LIN {X 0,Y 370.334,Z 1271.38,A -85,B 0,C 180,E1 17928.905,E2 17928.905} C_VEL
LIN {X 0,Y 369.324,Z 1281.028,A -85,B 0,C 180,E1 17925.869,E2 17925.869} C_VEL
LIN {X 0,Y 368.724,Z 1288.757,A -85,B 0,C 180,E1 17922.848,E2 17922.848} C_VEL
LIN {X 0,Y 368.382,Z 1295.019,A -85,B 0,C 180,E1 17919.688,E2 17919.688} C_VEL
LIN {X 0,Y 368.28,Z 1299.31,A -85,B 0,C 180,E1 17916.705,E2 17916.705} C_VEL
LIN {X 0,Y 368.262,Z 1302.013,A -85,B 0,C 180,E1 17913.737,E2 17913.737} C_VEL
LIN {X 0,Y 368.271,Z 1303.134,A -85,B 0,C 180,E1 17910.779,E2 17910.779} C_VEL
LIN {X 0,Y 368.275,Z 1302.722,A -85,B 0,C 180,E1 17907.667,E2 17907.667} C_VEL
LIN {X 0,Y 368.252,Z 1300.81,A -85,B 0,C 180,E1 17904.704,E2 17904.704} C_VEL
LIN {X 0,Y 368.291,Z 1297.252,A -85,B 0,C 180,E1 17901.728,E2 17901.728} C_VEL
LIN {X 0,Y 368.472,Z 1292.124,A -85,B 0,C 180,E1 17898.734,E2 17898.734} C_VEL
LIN {X 0,Y 368.884,Z 1285.33,A -85,B 0,C 180,E1 17895.721,E2 17895.721} C_VEL
LIN {X 0,Y 369.628,Z 1276.713,A -85,B 0,C 180,E1 17892.69,E2 17892.69} C_VEL
LIN {X 0,Y 370.897,Z 1266.188,A -85,B 0,C 180,E1 17889.486,E2 17889.486} C_VEL
LIN {X 0,Y 372.62,Z 1254.112,A -85,B 0,C 180,E1 17886.434,E2 17886.434} C_VEL
LIN {X 0,Y 374.842,Z 1240.532,A -85,B 0,C 180,E1 17883.548,E2 17883.548} C_VEL
LIN {X 0,Y 377.687,Z 1224.468,A -85,B 0,C 180,E1 17880.677,E2 17880.677} C_VEL
LIN {X 0,Y 380.995,Z 1206.604,A -85,B 0,C 180,E1 17877.988,E2 17877.988} C_VEL
LIN {X 0,Y 384.421,Z 1188.101,A -85,B 0,C 180,E1 17875.64,E2 17875.64} C_VEL
LIN {X 0,Y 387.844,Z 1169.342,A -85,B 0,C 180,E1 17873.635,E2 17873.635} C_VEL
LIN {X 0,Y 391.563,Z 1148.3,A -85,B 0,C 180,E1 17871.741,E2 17871.741} C_VEL
LIN {X 0,Y 394.879,Z 1128.554,A -85,B 0,C 180,E1 17870.258,E2 17870.258} C_VEL
LIN {X 0,Y 398.329,Z 1105.945,A -85,B 0,C 180,E1 17868.88,E2 17868.88} C_VEL
LIN {X 0,Y 401.441,Z 1082.847,A -85,B 0,C 180,E1 17867.777,E2 17867.777} C_VEL
LIN {X 0,Y 404.065,Z 1059.287,A -85,B 0,C 180,E1 17866.948,E2 17866.948} C_VEL
LIN {X 0,Y 405.779,Z 1035.371,A -85,B 0,C 180,E1 17866.328,E2 17866.328} C_VEL
LIN {X 0,Y 407.409,Z 1016.443,A -85,B 0,C 180,E1 17865.98,E2 17865.98} C_VEL
LIN {X 0,Y 408.442,Z 1008.559,A -85,B 0,C 180,E1 17865.858,E2 17865.858} C_VEL
LIN {X 0,Y 420.821,Z 978.098,A -85,B 0,C 180,E1 17864.422,E2 17864.422} C_VEL
LIN {X 0,Y 430.29,Z 959.013,A -85,B 0,C 180,E1 17863.726,E2 17863.726} C_VEL
LIN {X 0,Y 442.106,Z 935.256,A -85,B 0,C 180,E1 17862.901,E2 17862.901} C_VEL
LIN {X 0,Y 444.175,Z 931.152,A -85,B 0,C 180,E1 17862.767,E2 17862.767} C_VEL
LIN {X 0,Y 436.092,Z 918.557,A -85,B 0,C 180,E1 17860.801,E2 17860.801} C_VEL
LIN {X 0,Y 429.406,Z 903.824,A -85,B 0,C 180,E1 17858.696,E2 17858.696} C_VEL
LIN {X 0,Y 424.66,Z 887.722,A -85,B 0,C 180,E1 17856.595,E2 17856.595} C_VEL
LIN {X 0,Y 421.837,Z 870.153,A -85,B 0,C 180,E1 17854.505,E2 17854.505} C_VEL
LIN {X 0,Y 420.994,Z 850.406,A -85,B 0,C 180,E1 17852.382,E2 17852.382} C_VEL
LIN {X 0,Y 422.168,Z 830.506,A -85,B 0,C 180,E1 17850.449,E2 17850.449} C_VEL
LIN {X 0,Y 426.561,Z 800.035,A -85,B 0,C 180,E1 17847.804,E2 17847.804} C_VEL
LIN {X 0,Y 427.695,Z 792.967,A -85,B 0,C 180,E1 17847.196,E2 17847.196} C_VEL
LIN {X 0,Y 418.747,Z 775.54,A -85,B 0,C 180,E1 17843.649,E2 17843.649} C_VEL
LIN {X 0,Y 409.719,Z 758.616,A -85,B 0,C 180,E1 17839.828,E2 17839.828} C_VEL
LIN {X 0,Y 401.65,Z 744.073,A -85,B 0,C 180,E1 17836.189,E2 17836.189} C_VEL
LIN {X 0,Y 395.059,Z 732.588,A -85,B 0,C 180,E1 17833.017,E2 17833.017} C_VEL
LIN {X 0,Y 390.083,Z 723.936,A -85,B 0,C 180,E1 17830.485,E2 17830.485} C_VEL
LIN {X 0,Y 387.124,Z 718.9,A -85,B 0,C 180,E1 17828.915,E2 17828.915} C_VEL
LIN {X 0,Y 384.512,Z 714.317,A -85,B 0,C 180,E1 17827.47,E2 17827.47} C_VEL
LIN {X 0,Y 381.689,Z 709.437,A -85,B 0,C 180,E1 17825.863,E2 17825.863} C_VEL
LIN {X 0,Y 379.41,Z 705.573,A -85,B 0,C 180,E1 17824.534,E2 17824.534} C_VEL
LIN {X 0,Y 378.063,Z 703.576,A -85,B 0,C 180,E1 17823.791,E2 17823.791} C_VEL
LIN {X 0,Y 375.728,Z 699.193,A -85,B 0,C 180,E1 17822.287,E2 17822.287} C_VEL
LIN {X 0,Y 373.418,Z 695.781,A -85,B 0,C 180,E1 17820.92,E2 17820.92} C_VEL
LIN {X 0,Y 372.606,Z 693.864,A -85,B 0,C 180,E1 17820.307,E2 17820.307} C_VEL
LIN {X 0,Y 370.262,Z 690.693,A -85,B 0,C 180,E1 17818.917,E2 17818.917} C_VEL
LIN {X 0,Y 369.747,Z 688.673,A -85,B 0,C 180,E1 17818.295,E2 17818.295} C_VEL
LIN {X 0,Y 369.749,Z 688.674,A -85,B 0,C 180,E1 17814.102,E2 17814.102} C_VEL
LIN {X 0,Y 369.75,Z 688.677,A -85,B 0,C 180,E1 17809.876,E2 17809.876} C_VEL
LIN {X 0,Y 369.748,Z 688.678,A -85,B 0,C 180,E1 17805.754,E2 17805.754} C_VEL
LIN {X 0,Y 369.737,Z 688.666,A -85,B 0,C 180,E1 17801.654,E2 17801.654} C_VEL
LIN {X 0,Y 369.739,Z 688.667,A -85,B 0,C 180,E1 17797.586,E2 17797.586} C_VEL
LIN {X 0,Y 369.743,Z 688.647,A -85,B 0,C 180,E1 17793.5,E2 17793.5} C_VEL
LIN {X 0,Y 369.739,Z 688.661,A -85,B 0,C 180,E1 17789.674,E2 17789.674} C_VEL
LIN {X 0,Y 370.97,Z 692.001,A -85,B 0,C 180,E1 17788.99,E2 17788.99} C_VEL
LIN {X 0,Y 373.172,Z 694.719,A -85,B 0,C 180,E1 17788.14,E2 17788.14} C_VEL
LIN {X 0,Y 375.236,Z 698.459,A -85,B 0,C 180,E1 17787.254,E2 17787.254} C_VEL
LIN {X 0,Y 376.535,Z 700.304,A -85,B 0,C 180,E1 17786.766,E2 17786.766} C_VEL
LIN {X 0,Y 382.225,Z 710.075,A -85,B 0,C 180,E1 17784.498,E2 17784.498} C_VEL
LIN {X 0,Y 389.28,Z 723.15,A -85,B 0,C 180,E1 17781.756,E2 17781.756} C_VEL
LIN {X 0,Y 396.449,Z 737.875,A -85,B 0,C 180,E1 17779.025,E2 17779.025} C_VEL
LIN {X 0,Y 403.876,Z 755.101,A -85,B 0,C 180,E1 17776.215,E2 17776.215} C_VEL
LIN {X 0,Y 407.155,Z 763.877,A -85,B 0,C 180,E1 17774.938,E2 17774.938} C_VEL
LIN {X 0,Y 406.421,Z 778.004,A -85,B 0,C 180,E1 17773.911,E2 17773.911} C_VEL
LIN {X 0,Y 409.717,Z 805.43,A -85,B 0,C 180,E1 17772.811,E2 17772.811} C_VEL
LIN {X 0,Y 401.369,Z 1038.951,A -85,B 0,C 180,E1 17768.404,E2 17768.404} C_VEL
LIN {X 0,Y 400.003,Z 1059.693,A -85,B 0,C 180,E1 17767.771,E2 17767.771} C_VEL
LIN {X 0,Y 398.071,Z 1079.901,A -85,B 0,C 180,E1 17766.891,E2 17766.891} C_VEL
LIN {X 0,Y 395.711,Z 1098.998,A -85,B 0,C 180,E1 17765.798,E2 17765.798} C_VEL
LIN {X 0,Y 392.961,Z 1117.404,A -85,B 0,C 180,E1 17764.473,E2 17764.473} C_VEL
LIN {X 0,Y 389.794,Z 1135.566,A -85,B 0,C 180,E1 17762.854,E2 17762.854} C_VEL
LIN {X 0,Y 386.595,Z 1152.047,A -85,B 0,C 180,E1 17761.061,E2 17761.061} C_VEL
LIN {X 0,Y 383.311,Z 1167.686,A -85,B 0,C 180,E1 17759.023,E2 17759.023} C_VEL
LIN {X 0,Y 380.099,Z 1182.367,A -85,B 0,C 180,E1 17756.731,E2 17756.731} C_VEL
LIN {X 0,Y 377.097,Z 1195.87,A -85,B 0,C 180,E1 17754.202,E2 17754.202} C_VEL
LIN {X 0,Y 376.683,Z 1197.706,A -85,B 0,C 180,E1 17753.819,E2 17753.819} C_VEL
LIN {X 0,Y 374.766,Z 1202.283,A -85,B 0,C 180,E1 17752.903,E2 17752.903} C_VEL
LIN {X 0,Y 366.788,Z 1213.338,A -85,B 0,C 180,E1 17750.607,E2 17750.607} C_VEL
LIN {X 0,Y 365.037,Z 1217.109,A -85,B 0,C 180,E1 17749.588,E2 17749.588} C_VEL
LIN {X 0,Y 363.2,Z 1226.026,A -85,B 0,C 180,E1 17746.636,E2 17746.636} C_VEL
LIN {X 0,Y 361.799,Z 1233.817,A -85,B 0,C 180,E1 17743.398,E2 17743.398} C_VEL
LIN {X 0,Y 360.949,Z 1239.677,A -85,B 0,C 180,E1 17740.211,E2 17740.211} C_VEL
LIN {X 0,Y 360.49,Z 1243.91,A -85,B 0,C 180,E1 17737.009,E2 17737.009} C_VEL
LIN {X 0,Y 360.28,Z 1246.508,A -85,B 0,C 180,E1 17733.818,E2 17733.818} C_VEL
LIN {X 0,Y 360.214,Z 1247.557,A -85,B 0,C 180,E1 17730.635,E2 17730.635} C_VEL
LIN {X 0,Y 360.238,Z 1247.128,A -85,B 0,C 180,E1 17727.454,E2 17727.454} C_VEL
LIN {X 0,Y 360.371,Z 1245.21,A -85,B 0,C 180,E1 17724.267,E2 17724.267} C_VEL
LIN {X 0,Y 360.714,Z 1241.72,A -85,B 0,C 180,E1 17721.069,E2 17721.069} C_VEL
LIN {X 0,Y 361.39,Z 1236.528,A -85,B 0,C 180,E1 17717.861,E2 17717.861} C_VEL
LIN {X 0,Y 362.462,Z 1229.973,A -85,B 0,C 180,E1 17714.807,E2 17714.807} C_VEL
LIN {X 0,Y 364.176,Z 1221.194,A -85,B 0,C 180,E1 17711.594,E2 17711.594} C_VEL
LIN {X 0,Y 366.437,Z 1210.813,A -85,B 0,C 180,E1 17708.553,E2 17708.553} C_VEL
LIN {X 0,Y 369.026,Z 1199.594,A -85,B 0,C 180,E1 17705.849,E2 17705.849} C_VEL
LIN {X 0,Y 371.993,Z 1187.057,A -85,B 0,C 180,E1 17703.328,E2 17703.328} C_VEL
LIN {X 0,Y 375.48,Z 1172.083,A -85,B 0,C 180,E1 17700.836,E2 17700.836} C_VEL
LIN {X 0,Y 378.941,Z 1156.452,A -85,B 0,C 180,E1 17698.681,E2 17698.681} C_VEL
LIN {X 0,Y 382.302,Z 1140.187,A -85,B 0,C 180,E1 17696.816,E2 17696.816} C_VEL
LIN {X 0,Y 385.626,Z 1122.381,A -85,B 0,C 180,E1 17695.129,E2 17695.129} C_VEL
LIN {X 0,Y 388.618,Z 1104.067,A -85,B 0,C 180,E1 17693.718,E2 17693.718} C_VEL
LIN {X 0,Y 391.179,Z 1085.559,A -85,B 0,C 180,E1 17692.575,E2 17692.575} C_VEL
LIN {X 0,Y 393.361,Z 1065.157,A -85,B 0,C 180,E1 17691.604,E2 17691.604} C_VEL
LIN {X 0,Y 394.969,Z 1043.732,A -85,B 0,C 180,E1 17690.883,E2 17690.883} C_VEL
LIN {X 0,Y 396.204,Z 1013.325,A -85,B 0,C 180,E1 17690.248,E2 17690.248} C_VEL
LIN {X 0,Y 403.433,Z 816.76,A -85,B 0,C 180,E1 17686.515,E2 17686.515} C_VEL
LIN {X 0,Y 395.988,Z 779.414,A -85,B 0,C 180,E1 17684.495,E2 17684.495} C_VEL
LIN {X 0,Y 396.639,Z 768.209,A -85,B 0,C 180,E1 17683.237,E2 17683.237} C_VEL
LIN {X 0,Y 394.121,Z 760.718,A -85,B 0,C 180,E1 17681.853,E2 17681.853} C_VEL
LIN {X 0,Y 393.361,Z 760.544,A -85,B 0,C 180,E1 17681.642,E2 17681.642} C_VEL
LIN {X 0,Y 394.85,Z 764.717,A -85,B 0,C 180,E1 17680.898,E2 17680.898} C_VEL
LIN {X 0,Y 389.829,Z 803.215,A -85,B 0,C 180,E1 17676.8,E2 17676.8} C_VEL
LIN {X 0,Y 385.068,Z 843.255,A -85,B 0,C 180,E1 17672.602,E2 17672.602} C_VEL
LIN {X 0,Y 382.539,Z 867.952,A -85,B 0,C 180,E1 17670.081,E2 17670.081} C_VEL
LIN {X 0,Y 383.563,Z 877.843,A -85,B 0,C 180,E1 17669.684,E2 17669.684} C_VEL
LIN {X 0,Y 375.672,Z 1037.088,A -85,B 0,C 180,E1 17665.526,E2 17665.526} C_VEL
LIN {X 0,Y 374.898,Z 1054.189,A -85,B 0,C 180,E1 17664.838,E2 17664.838} C_VEL
LIN {X 0,Y 373.669,Z 1071.817,A -85,B 0,C 180,E1 17663.832,E2 17663.832} C_VEL
LIN {X 0,Y 372.206,Z 1088.344,A -85,B 0,C 180,E1 17662.591,E2 17662.591} C_VEL
LIN {X 0,Y 370.57,Z 1103.821,A -85,B 0,C 180,E1 17661.113,E2 17661.113} C_VEL
LIN {X 0,Y 368.793,Z 1118.857,A -85,B 0,C 180,E1 17659.315,E2 17659.315} C_VEL
LIN {X 0,Y 367.142,Z 1131.984,A -85,B 0,C 180,E1 17657.39,E2 17657.39} C_VEL
LIN {X 0,Y 365.594,Z 1143.989,A -85,B 0,C 180,E1 17655.222,E2 17655.222} C_VEL
LIN {X 0,Y 364.239,Z 1154.622,A -85,B 0,C 180,E1 17652.847,E2 17652.847} C_VEL
LIN {X 0,Y 363.188,Z 1163.735,A -85,B 0,C 180,E1 17650.309,E2 17650.309} C_VEL
LIN {X 0,Y 362.494,Z 1170.776,A -85,B 0,C 180,E1 17647.768,E2 17647.768} C_VEL
LIN {X 0,Y 362.034,Z 1176.672,A -85,B 0,C 180,E1 17644.912,E2 17644.912} C_VEL
LIN {X 0,Y 361.881,Z 1180.442,A -85,B 0,C 180,E1 17642.217,E2 17642.217} C_VEL
LIN {X 0,Y 361.917,Z 1182.564,A -85,B 0,C 180,E1 17639.367,E2 17639.367} C_VEL
LIN {X 0,Y 362.162,Z 1182.94,A -85,B 0,C 180,E1 17636.518,E2 17636.518} C_VEL
LIN {X 0,Y 362.626,Z 1181.617,A -85,B 0,C 180,E1 17633.827,E2 17633.827} C_VEL
LIN {X 0,Y 363.414,Z 1178.412,A -85,B 0,C 180,E1 17630.978,E2 17630.978} C_VEL
LIN {X 0,Y 364.517,Z 1173.647,A -85,B 0,C 180,E1 17628.289,E2 17628.289} C_VEL
LIN {X 0,Y 366.041,Z 1166.884,A -85,B 0,C 180,E1 17625.607,E2 17625.607} C_VEL
LIN {X 0,Y 367.931,Z 1158.574,A -85,B 0,C 180,E1 17623.096,E2 17623.096} C_VEL
LIN {X 0,Y 370.08,Z 1148.58,A -85,B 0,C 180,E1 17620.755,E2 17620.755} C_VEL
LIN {X 0,Y 372.266,Z 1137.95,A -85,B 0,C 180,E1 17618.741,E2 17618.741} C_VEL
LIN {X 0,Y 374.503,Z 1125.805,A -85,B 0,C 180,E1 17616.892,E2 17616.892} C_VEL
LIN {X 0,Y 376.769,Z 1112.27,A -85,B 0,C 180,E1 17615.21,E2 17615.21} C_VEL
LIN {X 0,Y 379.043,Z 1095.883,A -85,B 0,C 180,E1 17613.61,E2 17613.61} C_VEL
LIN {X 0,Y 380.683,Z 1080.836,A -85,B 0,C 180,E1 17612.467,E2 17612.467} C_VEL
LIN {X 0,Y 382.09,Z 1064.158,A -85,B 0,C 180,E1 17611.495,E2 17611.495} C_VEL
LIN {X 0,Y 385.237,Z 1037.1,A -85,B 0,C 180,E1 17610.154,E2 17610.154} C_VEL
LIN {X 0,Y 394.185,Z 989.779,A -85,B 0,C 180,E1 17607.986,E2 17607.986} C_VEL
LIN {X 0,Y 405.123,Z 935.467,A -85,B 0,C 180,E1 17605.776,E2 17605.776} C_VEL
LIN {X 0,Y 406.823,Z 928.336,A -85,B 0,C 180,E1 17605.494,E2 17605.494} C_VEL
LIN {X 0,Y 417.353,Z 912.085,A -85,B 0,C 180,E1 17604.482,E2 17604.482} C_VEL
LIN {X 0,Y 423.503,Z 903.048,A -85,B 0,C 180,E1 17603.827,E2 17603.827} C_VEL
LIN {X 0,Y 426.01,Z 899.819,A -85,B 0,C 180,E1 17603.301,E2 17603.301} C_VEL
LIN {X 0,Y 424.14,Z 907.115,A -85,B 0,C 180,E1 17601.504,E2 17601.504} C_VEL
LIN {X 0,Y 424.485,Z 914.511,A -85,B 0,C 180,E1 17599.745,E2 17599.745} C_VEL
LIN {X 0,Y 427.026,Z 922.456,A -85,B 0,C 180,E1 17597.96,E2 17597.96} C_VEL
LIN {X 0,Y 430.407,Z 928.617,A -85,B 0,C 180,E1 17596.646,E2 17596.646} C_VEL
LIN {X 0,Y 420.892,Z 947.99,A -85,B 0,C 180,E1 17595.97,E2 17595.97} C_VEL
LIN {X 0,Y 409.338,Z 971.916,A -85,B 0,C 180,E1 17595.102,E2 17595.102} C_VEL
LIN {X 0,Y 407.173,Z 977.442,A -85,B 0,C 180,E1 17594.891,E2 17594.891} C_VEL
LIN {X 0,Y 403.741,Z 996.518,A -85,B 0,C 180,E1 17594.623,E2 17594.623} C_VEL
LIN {X 0,Y 399.024,Z 1022.37,A -85,B 0,C 180,E1 17594.225,E2 17594.225} C_VEL
LIN {X 0,Y 396.381,Z 1040.88,A -85,B 0,C 180,E1 17593.63,E2 17593.63} C_VEL
LIN {X 0,Y 392.042,Z 1070.576,A -85,B 0,C 180,E1 17592.381,E2 17592.381} C_VEL
LIN {X 0,Y 387.903,Z 1096.54,A -85,B 0,C 180,E1 17590.996,E2 17590.996} C_VEL
LIN {X 0,Y 383.805,Z 1122.59,A -85,B 0,C 180,E1 17589.276,E2 17589.276} C_VEL
LIN {X 0,Y 379.789,Z 1149.026,A -85,B 0,C 180,E1 17587.208,E2 17587.208} C_VEL
LIN {X 0,Y 377.55,Z 1169.051,A -85,B 0,C 180,E1 17585.608,E2 17585.608} C_VEL
LIN {X 0,Y 375.105,Z 1187.196,A -85,B 0,C 180,E1 17583.856,E2 17583.856} C_VEL
LIN {X 0,Y 372.581,Z 1204.537,A -85,B 0,C 180,E1 17581.849,E2 17581.849} C_VEL
LIN {X 0,Y 370.039,Z 1220.672,A -85,B 0,C 180,E1 17579.636,E2 17579.636} C_VEL
LIN {X 0,Y 367.548,Z 1236.156,A -85,B 0,C 180,E1 17577.108,E2 17577.108} C_VEL
LIN {X 0,Y 365.512,Z 1249.285,A -85,B 0,C 180,E1 17574.57,E2 17574.57} C_VEL
LIN {X 0,Y 363.66,Z 1261.967,A -85,B 0,C 180,E1 17571.674,E2 17571.674} C_VEL
LIN {X 0,Y 362.251,Z 1272.901,A -85,B 0,C 180,E1 17568.674,E2 17568.674} C_VEL
LIN {X 0,Y 361.25,Z 1282.119,A -85,B 0,C 180,E1 17565.596,E2 17565.596} C_VEL
LIN {X 0,Y 360.683,Z 1289.596,A -85,B 0,C 180,E1 17562.488,E2 17562.488} C_VEL
LIN {X 0,Y 360.371,Z 1295.202,A -85,B 0,C 180,E1 17559.422,E2 17559.422} C_VEL
LIN {X 0,Y 360.293,Z 1299.202,A -85,B 0,C 180,E1 17556.374,E2 17556.374} C_VEL
LIN {X 0,Y 360.282,Z 1301.681,A -85,B 0,C 180,E1 17553.342,E2 17553.342} C_VEL
LIN {X 0,Y 360.297,Z 1302.595,A -85,B 0,C 180,E1 17550.319,E2 17550.319} C_VEL
LIN {X 0,Y 360.286,Z 1301.969,A -85,B 0,C 180,E1 17547.297,E2 17547.297} C_VEL
LIN {X 0,Y 360.267,Z 1299.87,A -85,B 0,C 180,E1 17544.267,E2 17544.267} C_VEL
LIN {X 0,Y 360.317,Z 1296.202,A -85,B 0,C 180,E1 17541.222,E2 17541.222} C_VEL
LIN {X 0,Y 360.532,Z 1290.87,A -85,B 0,C 180,E1 17538.158,E2 17538.158} C_VEL
LIN {X 0,Y 361.041,Z 1283.439,A -85,B 0,C 180,E1 17534.912,E2 17534.912} C_VEL
LIN {X 0,Y 361.915,Z 1274.491,A -85,B 0,C 180,E1 17531.81,E2 17531.81} C_VEL
LIN {X 0,Y 363.181,Z 1264.14,A -85,B 0,C 180,E1 17528.861,E2 17528.861} C_VEL
LIN {X 0,Y 365.064,Z 1251.734,A -85,B 0,C 180,E1 17525.744,E2 17525.744} C_VEL
LIN {X 0,Y 367.443,Z 1237.859,A -85,B 0,C 180,E1 17522.798,E2 17522.798} C_VEL
LIN {X 0,Y 370.298,Z 1222.447,A -85,B 0,C 180,E1 17520.032,E2 17520.032} C_VEL
LIN {X 0,Y 373.687,Z 1204.93,A -85,B 0,C 180,E1 17517.376,E2 17517.376} C_VEL
LIN {X 0,Y 377.164,Z 1186.99,A -85,B 0,C 180,E1 17515.068,E2 17515.068} C_VEL
LIN {X 0,Y 380.722,Z 1168.184,A -85,B 0,C 180,E1 17513.031,E2 17513.031} C_VEL
LIN {X 0,Y 384.556,Z 1147.378,A -85,B 0,C 180,E1 17511.134,E2 17511.134} C_VEL
LIN {X 0,Y 388.053,Z 1127.311,A -85,B 0,C 180,E1 17509.609,E2 17509.609} C_VEL
LIN {X 0,Y 391.691,Z 1104.318,A -85,B 0,C 180,E1 17508.191,E2 17508.191} C_VEL
LIN {X 0,Y 394.935,Z 1081.232,A -85,B 0,C 180,E1 17507.084,E2 17507.084} C_VEL
LIN {X 0,Y 397.625,Z 1057.81,A -85,B 0,C 180,E1 17506.252,E2 17506.252} C_VEL
LIN {X 0,Y 399.394,Z 1033.97,A -85,B 0,C 180,E1 17505.622,E2 17505.622} C_VEL
LIN {X 0,Y 401.317,Z 1013.867,A -85,B 0,C 180,E1 17505.26,E2 17505.26} C_VEL
LIN {X 0,Y 402.28,Z 1007.289,A -85,B 0,C 180,E1 17505.151,E2 17505.151} C_VEL
LIN {X 0,Y 414.92,Z 976.742,A -85,B 0,C 180,E1 17503.704,E2 17503.704} C_VEL
LIN {X 0,Y 424.534,Z 957.541,A -85,B 0,C 180,E1 17503.007,E2 17503.007} C_VEL
LIN {X 0,Y 436.362,Z 933.76,A -85,B 0,C 180,E1 17502.172,E2 17502.172} C_VEL
LIN {X 0,Y 428.84,Z 921.197,A -85,B 0,C 180,E1 17500.228,E2 17500.228} C_VEL
LIN {X 0,Y 422.391,Z 906.03,A -85,B 0,C 180,E1 17498.071,E2 17498.071} C_VEL
LIN {X 0,Y 417.987,Z 889.853,A -85,B 0,C 180,E1 17495.962,E2 17495.962} C_VEL
LIN {X 0,Y 415.477,Z 872.42,A -85,B 0,C 180,E1 17493.877,E2 17493.877} C_VEL
LIN {X 0,Y 414.883,Z 852.273,A -85,B 0,C 180,E1 17491.693,E2 17491.693} C_VEL
LIN {X 0,Y 416.372,Z 830.958,A -85,B 0,C 180,E1 17489.625,E2 17489.625} C_VEL
LIN {X 0,Y 421.545,Z 797.164,A -85,B 0,C 180,E1 17486.672,E2 17486.672} C_VEL
LIN {X 0,Y 413.058,Z 780.548,A -85,B 0,C 180,E1 17483.238,E2 17483.238} C_VEL
LIN {X 0,Y 404.386,Z 764.152,A -85,B 0,C 180,E1 17479.499,E2 17479.499} C_VEL
LIN {X 0,Y 396.616,Z 750.067,A -85,B 0,C 180,E1 17475.949,E2 17475.949} C_VEL
LIN {X 0,Y 388.955,Z 736.37,A -85,B 0,C 180,E1 17472.168,E2 17472.168} C_VEL
LIN {X 0,Y 382.323,Z 725.17,A -85,B 0,C 180,E1 17468.724,E2 17468.724} C_VEL
LIN {X 0,Y 379.43,Z 720.187,A -85,B 0,C 180,E1 17467.114,E2 17467.114} C_VEL
LIN {X 0,Y 376.591,Z 715.31,A -85,B 0,C 180,E1 17465.484,E2 17465.484} C_VEL
LIN {X 0,Y 373.763,Z 710.423,A -85,B 0,C 180,E1 17463.802,E2 17463.802} C_VEL
LIN {X 0,Y 371.379,Z 706.208,A -85,B 0,C 180,E1 17462.314,E2 17462.314} C_VEL
LIN {X 0,Y 368.581,Z 701.852,A -85,B 0,C 180,E1 17460.621,E2 17460.621} C_VEL
LIN {X 0,Y 367.696,Z 700.08,A -85,B 0,C 180,E1 17460,E2 17460} C_VEL
LIN {X 0,Y 365.419,Z 696.703,A -85,B 0,C 180,E1 17458.589,E2 17458.589} C_VEL
LIN {X 0,Y 364.65,Z 694.844,A -85,B 0,C 180,E1 17457.957,E2 17457.957} C_VEL
LIN {X 0,Y 362.53,Z 692.14,A -85,B 0,C 180,E1 17456.679,E2 17456.679} C_VEL
LIN {X 0,Y 361.799,Z 689.663,A -85,B 0,C 180,E1 17455.879,E2 17455.879} C_VEL
LIN {X 0,Y 361.805,Z 689.663,A -85,B 0,C 180,E1 17451.737,E2 17451.737} C_VEL
LIN {X 0,Y 361.81,Z 689.666,A -85,B 0,C 180,E1 17447.552,E2 17447.552} C_VEL
LIN {X 0,Y 361.808,Z 689.665,A -85,B 0,C 180,E1 17443.462,E2 17443.462} C_VEL
LIN {X 0,Y 361.816,Z 689.664,A -85,B 0,C 180,E1 17439.115,E2 17439.115} C_VEL
LIN {X 0,Y 361.806,Z 689.668,A -85,B 0,C 180,E1 17434.987,E2 17434.987} C_VEL
LIN {X 0,Y 361.81,Z 689.637,A -85,B 0,C 180,E1 17431.619,E2 17431.619} C_VEL
LIN {X 0,Y 362.81,Z 692.621,A -85,B 0,C 180,E1 17430.985,E2 17430.985} C_VEL
LIN {X 0,Y 365.352,Z 695.631,A -85,B 0,C 180,E1 17429.946,E2 17429.946} C_VEL
LIN {X 0,Y 367.29,Z 699.312,A -85,B 0,C 180,E1 17429.035,E2 17429.035} C_VEL
LIN {X 0,Y 368.771,Z 701.272,A -85,B 0,C 180,E1 17428.447,E2 17428.447} C_VEL
LIN {X 0,Y 371.173,Z 705.302,A -85,B 0,C 180,E1 17427.401,E2 17427.401} C_VEL
LIN {X 0,Y 377.304,Z 715.803,A -85,B 0,C 180,E1 17424.896,E2 17424.896} C_VEL
LIN {X 0,Y 384.252,Z 728.889,A -85,B 0,C 180,E1 17422.113,E2 17422.113} C_VEL
LIN {X 0,Y 391.319,Z 743.645,A -85,B 0,C 180,E1 17419.341,E2 17419.341} C_VEL
LIN {X 0,Y 398.456,Z 760.469,A -85,B 0,C 180,E1 17416.563,E2 17416.563} C_VEL
LIN {X 0,Y 401.144,Z 767.307,A -85,B 0,C 180,E1 17415.541,E2 17415.541} C_VEL
LIN {X 0,Y 400.564,Z 778.616,A -85,B 0,C 180,E1 17414.72,E2 17414.72} C_VEL
LIN {X 0,Y 403.859,Z 806.865,A -85,B 0,C 180,E1 17413.563,E2 17413.563} C_VEL
LIN {X 0,Y 395.135,Z 1039.668,A -85,B 0,C 180,E1 17409.119,E2 17409.119} C_VEL
LIN {X 0,Y 393.72,Z 1060.288,A -85,B 0,C 180,E1 17408.481,E2 17408.481} C_VEL
LIN {X 0,Y 391.63,Z 1081.191,A -85,B 0,C 180,E1 17407.556,E2 17407.556} C_VEL
LIN {X 0,Y 389.087,Z 1100.679,A -85,B 0,C 180,E1 17406.413,E2 17406.413} C_VEL
LIN {X 0,Y 386.237,Z 1118.798,A -85,B 0,C 180,E1 17405.077,E2 17405.077} C_VEL
LIN {X 0,Y 382.934,Z 1136.929,A -85,B 0,C 180,E1 17403.43,E2 17403.43} C_VEL
LIN {X 0,Y 379.467,Z 1153.947,A -85,B 0,C 180,E1 17401.535,E2 17401.535} C_VEL
LIN {X 0,Y 375.979,Z 1169.684,A -85,B 0,C 180,E1 17399.419,E2 17399.419} C_VEL
LIN {X 0,Y 372.697,Z 1183.874,A -85,B 0,C 180,E1 17397.133,E2 17397.133} C_VEL
LIN {X 0,Y 369.628,Z 1196.944,A -85,B 0,C 180,E1 17394.618,E2 17394.618} C_VEL
LIN {X 0,Y 366.923,Z 1208.631,A -85,B 0,C 180,E1 17391.92,E2 17391.92} C_VEL
LIN {X 0,Y 365.037,Z 1217.109,A -85,B 0,C 180,E1 17389.588,E2 17389.588} C_VEL
LIN {X 0,Y 363.336,Z 1220.757,A -85,B 0,C 180,E1 17388.543,E2 17388.543} C_VEL
LIN {X 0,Y 355.548,Z 1229.785,A -85,B 0,C 180,E1 17385.732,E2 17385.732} C_VEL
LIN {X 0,Y 354.378,Z 1232.205,A -85,B 0,C 180,E1 17384.751,E2 17384.751} C_VEL
LIN {X 0,Y 353.31,Z 1238.42,A -85,B 0,C 180,E1 17381.59,E2 17381.59} C_VEL
LIN {X 0,Y 352.675,Z 1243.194,A -85,B 0,C 180,E1 17378.313,E2 17378.313} C_VEL
LIN {X 0,Y 352.365,Z 1246.365,A -85,B 0,C 180,E1 17375.046,E2 17375.046} C_VEL
LIN {X 0,Y 352.249,Z 1248.015,A -85,B 0,C 180,E1 17371.789,E2 17371.789} C_VEL
LIN {X 0,Y 352.24,Z 1248.094,A -85,B 0,C 180,E1 17368.698,E2 17368.698} C_VEL
LIN {X 0,Y 352.333,Z 1246.751,A -85,B 0,C 180,E1 17365.442,E2 17365.442} C_VEL
LIN {X 0,Y 352.598,Z 1243.897,A -85,B 0,C 180,E1 17362.176,E2 17362.176} C_VEL
LIN {X 0,Y 353.177,Z 1239.448,A -85,B 0,C 180,E1 17358.9,E2 17358.9} C_VEL
LIN {X 0,Y 354.268,Z 1232.889,A -85,B 0,C 180,E1 17355.452,E2 17355.452} C_VEL
LIN {X 0,Y 355.898,Z 1224.699,A -85,B 0,C 180,E1 17352.168,E2 17352.168} C_VEL
LIN {X 0,Y 357.954,Z 1215.506,A -85,B 0,C 180,E1 17349.222,E2 17349.222} C_VEL
LIN {X 0,Y 360.624,Z 1204.375,A -85,B 0,C 180,E1 17346.295,E2 17346.295} C_VEL
LIN {X 0,Y 363.755,Z 1191.754,A -85,B 0,C 180,E1 17343.557,E2 17343.557} C_VEL
LIN {X 0,Y 367.123,Z 1178.085,A -85,B 0,C 180,E1 17341.09,E2 17341.09} C_VEL
LIN {X 0,Y 370.751,Z 1162.946,A -85,B 0,C 180,E1 17338.815,E2 17338.815} C_VEL
LIN {X 0,Y 374.358,Z 1146.839,A -85,B 0,C 180,E1 17336.802,E2 17336.802} C_VEL
LIN {X 0,Y 377.876,Z 1129.474,A -85,B 0,C 180,E1 17335.018,E2 17335.018} C_VEL
LIN {X 0,Y 381.026,Z 1111.837,A -85,B 0,C 180,E1 17333.532,E2 17333.532} C_VEL
LIN {X 0,Y 383.894,Z 1093.135,A -85,B 0,C 180,E1 17332.261,E2 17332.261} C_VEL
LIN {X 0,Y 386.353,Z 1073.22,A -85,B 0,C 180,E1 17331.204,E2 17331.204} C_VEL
LIN {X 0,Y 388.177,Z 1053.47,A -85,B 0,C 180,E1 17330.423,E2 17330.423} C_VEL
LIN {X 0,Y 389.395,Z 1032.495,A -85,B 0,C 180,E1 17329.859,E2 17329.859} C_VEL
LIN {X 0,Y 397.671,Z 818.699,A -85,B 0,C 180,E1 17325.76,E2 17325.76} C_VEL
LIN {X 0,Y 390.082,Z 780.319,A -85,B 0,C 180,E1 17323.642,E2 17323.642} C_VEL
LIN {X 0,Y 390.524,Z 772.221,A -85,B 0,C 180,E1 17322.725,E2 17322.725} C_VEL
LIN {X 0,Y 388.925,Z 767.404,A -85,B 0,C 180,E1 17321.846,E2 17321.846} C_VEL
LIN {X 0,Y 387.838,Z 767.062,A -85,B 0,C 180,E1 17321.594,E2 17321.594} C_VEL
LIN {X 0,Y 388.24,Z 768.475,A -85,B 0,C 180,E1 17321.354,E2 17321.354} C_VEL
LIN {X 0,Y 382.997,Z 806.806,A -85,B 0,C 180,E1 17317.227,E2 17317.227} C_VEL
LIN {X 0,Y 378.087,Z 846.622,A -85,B 0,C 180,E1 17313.009,E2 17313.009} C_VEL
LIN {X 0,Y 375.688,Z 868.914,A -85,B 0,C 180,E1 17310.705,E2 17310.705} C_VEL
LIN {X 0,Y 376.687,Z 879.138,A -85,B 0,C 180,E1 17310.287,E2 17310.287} C_VEL
LIN {X 0,Y 368.367,Z 1037.296,A -85,B 0,C 180,E1 17306.029,E2 17306.029} C_VEL
LIN {X 0,Y 367.511,Z 1055.436,A -85,B 0,C 180,E1 17305.286,E2 17305.286} C_VEL
LIN {X 0,Y 366.228,Z 1073.122,A -85,B 0,C 180,E1 17304.252,E2 17304.252} C_VEL
LIN {X 0,Y 364.719,Z 1089.491,A -85,B 0,C 180,E1 17302.996,E2 17302.996} C_VEL
LIN {X 0,Y 363.023,Z 1104.981,A -85,B 0,C 180,E1 17301.489,E2 17301.489} C_VEL
LIN {X 0,Y 361.178,Z 1120.029,A -85,B 0,C 180,E1 17299.655,E2 17299.655} C_VEL
LIN {X 0,Y 359.433,Z 1133.42,A -85,B 0,C 180,E1 17297.651,E2 17297.651} C_VEL
LIN {X 0,Y 357.799,Z 1145.602,A -85,B 0,C 180,E1 17295.396,E2 17295.396} C_VEL
LIN {X 0,Y 356.403,Z 1156.212,A -85,B 0,C 180,E1 17292.97,E2 17292.97} C_VEL
LIN {X 0,Y 355.321,Z 1165.286,A -85,B 0,C 180,E1 17290.376,E2 17290.376} C_VEL
LIN {X 0,Y 354.571,Z 1172.685,A -85,B 0,C 180,E1 17287.616,E2 17287.616} C_VEL
LIN {X 0,Y 354.145,Z 1178.194,A -85,B 0,C 180,E1 17284.859,E2 17284.859} C_VEL
LIN {X 0,Y 353.991,Z 1181.934,A -85,B 0,C 180,E1 17282.105,E2 17282.105} C_VEL
LIN {X 0,Y 354.045,Z 1183.986,A -85,B 0,C 180,E1 17279.353,E2 17279.353} C_VEL
LIN {X 0,Y 354.317,Z 1184.454,A -85,B 0,C 180,E1 17276.441,E2 17276.441} C_VEL
LIN {X 0,Y 354.828,Z 1183.227,A -85,B 0,C 180,E1 17273.691,E2 17273.691} C_VEL
LIN {X 0,Y 355.688,Z 1180.132,A -85,B 0,C 180,E1 17270.78,E2 17270.78} C_VEL
LIN {X 0,Y 356.888,Z 1175.482,A -85,B 0,C 180,E1 17268.035,E2 17268.035} C_VEL
LIN {X 0,Y 358.533,Z 1168.859,A -85,B 0,C 180,E1 17265.299,E2 17265.299} C_VEL
LIN {X 0,Y 360.56,Z 1160.705,A -85,B 0,C 180,E1 17262.74,E2 17262.74} C_VEL
LIN {X 0,Y 362.861,Z 1150.917,A -85,B 0,C 180,E1 17260.357,E2 17260.357} C_VEL
LIN {X 0,Y 365.187,Z 1140.49,A -85,B 0,C 180,E1 17258.308,E2 17258.308} C_VEL
LIN {X 0,Y 367.659,Z 1128.326,A -85,B 0,C 180,E1 17256.378,E2 17256.378} C_VEL
LIN {X 0,Y 370.231,Z 1114.241,A -85,B 0,C 180,E1 17254.571,E2 17254.571} C_VEL
LIN {X 0,Y 372.683,Z 1098.347,A -85,B 0,C 180,E1 17252.964,E2 17252.964} C_VEL
LIN {X 0,Y 374.75,Z 1081.54,A -85,B 0,C 180,E1 17251.646,E2 17251.646} C_VEL
LIN {X 0,Y 376.915,Z 1060.18,A -85,B 0,C 180,E1 17250.392,E2 17250.392} C_VEL
LIN {X 0,Y 381.485,Z 1032.197,A -85,B 0,C 180,E1 17248.914,E2 17248.914} C_VEL
LIN {X 0,Y 396.211,Z 966.404,A -85,B 0,C 180,E1 17245.885,E2 17245.885} C_VEL
LIN {X 0,Y 403.777,Z 933.037,A -85,B 0,C 180,E1 17244.557,E2 17244.557} C_VEL
LIN {X 0,Y 414.588,Z 917.007,A -85,B 0,C 180,E1 17243.611,E2 17243.611} C_VEL
LIN {X 0,Y 420.586,Z 908.618,A -85,B 0,C 180,E1 17243.014,E2 17243.014} C_VEL
LIN {X 0,Y 419.235,Z 915.921,A -85,B 0,C 180,E1 17241.153,E2 17241.153} C_VEL
LIN {X 0,Y 420.168,Z 923.512,A -85,B 0,C 180,E1 17239.306,E2 17239.306} C_VEL
LIN {X 0,Y 423.571,Z 931.932,A -85,B 0,C 180,E1 17237.384,E2 17237.384} C_VEL
LIN {X 0,Y 411.804,Z 955.636,A -85,B 0,C 180,E1 17236.55,E2 17236.55} C_VEL
LIN {X 0,Y 403.611,Z 973.145,A -85,B 0,C 180,E1 17235.911,E2 17235.911} C_VEL
LIN {X 0,Y 399.523,Z 994.974,A -85,B 0,C 180,E1 17235.584,E2 17235.584} C_VEL
LIN {X 0,Y 394.364,Z 1021.131,A -85,B 0,C 180,E1 17235.17,E2 17235.17} C_VEL
LIN {X 0,Y 391.542,Z 1037.858,A -85,B 0,C 180,E1 17234.626,E2 17234.626} C_VEL
LIN {X 0,Y 386.727,Z 1067.362,A -85,B 0,C 180,E1 17233.349,E2 17233.349} C_VEL
LIN {X 0,Y 381.988,Z 1094.38,A -85,B 0,C 180,E1 17231.872,E2 17231.872} C_VEL
LIN {X 0,Y 377.508,Z 1120.116,A -85,B 0,C 180,E1 17230.134,E2 17230.134} C_VEL
LIN {X 0,Y 374.033,Z 1141.292,A -85,B 0,C 180,E1 17228.473,E2 17228.473} C_VEL
LIN {X 0,Y 371.843,Z 1160.539,A -85,B 0,C 180,E1 17227.037,E2 17227.037} C_VEL
LIN {X 0,Y 369.304,Z 1179.452,A -85,B 0,C 180,E1 17225.313,E2 17225.313} C_VEL
LIN {X 0,Y 366.58,Z 1197.406,A -85,B 0,C 180,E1 17223.34,E2 17223.34} C_VEL
LIN {X 0,Y 363.739,Z 1214.374,A -85,B 0,C 180,E1 17221.117,E2 17221.117} C_VEL
LIN {X 0,Y 361.116,Z 1229.829,A -85,B 0,C 180,E1 17218.711,E2 17218.711} C_VEL
LIN {X 0,Y 358.753,Z 1243.873,A -85,B 0,C 180,E1 17216.127,E2 17216.127} C_VEL
LIN {X 0,Y 356.622,Z 1256.842,A -85,B 0,C 180,E1 17213.287,E2 17213.287} C_VEL
LIN {X 0,Y 355.014,Z 1267.755,A -85,B 0,C 180,E1 17210.441,E2 17210.441} C_VEL
LIN {X 0,Y 353.736,Z 1277.874,A -85,B 0,C 180,E1 17207.266,E2 17207.266} C_VEL
LIN {X 0,Y 352.924,Z 1286.038,A -85,B 0,C 180,E1 17204.102,E2 17204.102} C_VEL
LIN {X 0,Y 352.49,Z 1292.449,A -85,B 0,C 180,E1 17200.956,E2 17200.956} C_VEL
LIN {X 0,Y 352.323,Z 1297.107,A -85,B 0,C 180,E1 17197.83,E2 17197.83} C_VEL
LIN {X 0,Y 352.298,Z 1300.196,A -85,B 0,C 180,E1 17194.722,E2 17194.722} C_VEL
LIN {X 0,Y 352.311,Z 1301.794,A -85,B 0,C 180,E1 17191.627,E2 17191.627} C_VEL
LIN {X 0,Y 352.314,Z 1301.843,A -85,B 0,C 180,E1 17188.7,E2 17188.7} C_VEL
LIN {X 0,Y 352.3,Z 1300.435,A -85,B 0,C 180,E1 17185.606,E2 17185.606} C_VEL
LIN {X 0,Y 352.288,Z 1297.536,A -85,B 0,C 180,E1 17182.499,E2 17182.499} C_VEL
LIN {X 0,Y 352.427,Z 1292.986,A -85,B 0,C 180,E1 17179.374,E2 17179.374} C_VEL
LIN {X 0,Y 352.783,Z 1286.775,A -85,B 0,C 180,E1 17176.228,E2 17176.228} C_VEL
LIN {X 0,Y 353.566,Z 1278.342,A -85,B 0,C 180,E1 17172.897,E2 17172.897} C_VEL
LIN {X 0,Y 354.758,Z 1268.331,A -85,B 0,C 180,E1 17169.717,E2 17169.717} C_VEL
LIN {X 0,Y 356.28,Z 1257.547,A -85,B 0,C 180,E1 17166.866,E2 17166.866} C_VEL
LIN {X 0,Y 359.211,Z 1239.829,A -85,B 0,C 180,E1 17162.962,E2 17162.962} C_VEL
LIN {X 0,Y 362.096,Z 1224.778,A -85,B 0,C 180,E1 17160.117,E2 17160.117} C_VEL
LIN {X 0,Y 365.28,Z 1208.831,A -85,B 0,C 180,E1 17157.555,E2 17157.555} C_VEL
LIN {X 0,Y 368.87,Z 1190.972,A -85,B 0,C 180,E1 17155.116,E2 17155.116} C_VEL
LIN {X 0,Y 372.947,Z 1170.473,A -85,B 0,C 180,E1 17152.773,E2 17152.773} C_VEL
LIN {X 0,Y 376.682,Z 1151.319,A -85,B 0,C 180,E1 17150.92,E2 17150.92} C_VEL
LIN {X 0,Y 380.714,Z 1129.219,A -85,B 0,C 180,E1 17149.162,E2 17149.162} C_VEL
LIN {X 0,Y 384.378,Z 1107.215,A -85,B 0,C 180,E1 17147.747,E2 17147.747} C_VEL
LIN {X 0,Y 387.856,Z 1083.771,A -85,B 0,C 180,E1 17146.556,E2 17146.556} C_VEL
LIN {X 0,Y 390.786,Z 1060.559,A -85,B 0,C 180,E1 17145.671,E2 17145.671} C_VEL
LIN {X 0,Y 392.721,Z 1037.234,A -85,B 0,C 180,E1 17145.018,E2 17145.018} C_VEL
LIN {X 0,Y 394.467,Z 1017.593,A -85,B 0,C 180,E1 17144.622,E2 17144.622} C_VEL
LIN {X 0,Y 396.007,Z 1006.407,A -85,B 0,C 180,E1 17144.448,E2 17144.448} C_VEL
LIN {X 0,Y 408.759,Z 975.981,A -85,B 0,C 180,E1 17142.999,E2 17142.999} C_VEL
LIN {X 0,Y 418.858,Z 955.991,A -85,B 0,C 180,E1 17142.27,E2 17142.27} C_VEL
LIN {X 0,Y 428.629,Z 936.28,A -85,B 0,C 180,E1 17141.555,E2 17141.555} C_VEL
LIN {X 0,Y 420.795,Z 921.991,A -85,B 0,C 180,E1 17139.377,E2 17139.377} C_VEL
LIN {X 0,Y 414.797,Z 906.1,A -85,B 0,C 180,E1 17137.144,E2 17137.144} C_VEL
LIN {X 0,Y 410.886,Z 889.19,A -85,B 0,C 180,E1 17134.964,E2 17134.964} C_VEL
LIN {X 0,Y 408.902,Z 870.761,A -85,B 0,C 180,E1 17132.793,E2 17132.793} C_VEL
LIN {X 0,Y 408.899,Z 850.226,A -85,B 0,C 180,E1 17130.604,E2 17130.604} C_VEL
LIN {X 0,Y 411.27,Z 826.608,A -85,B 0,C 180,E1 17128.351,E2 17128.351} C_VEL
LIN {X 0,Y 415.441,Z 801.34,A -85,B 0,C 180,E1 17126.131,E2 17126.131} C_VEL
LIN {X 0,Y 407.35,Z 785.506,A -85,B 0,C 180,E1 17122.818,E2 17122.818} C_VEL
LIN {X 0,Y 398.991,Z 769.641,A -85,B 0,C 180,E1 17119.164,E2 17119.164} C_VEL
LIN {X 0,Y 391.249,Z 755.548,A -85,B 0,C 180,E1 17115.565,E2 17115.565} C_VEL
LIN {X 0,Y 383.896,Z 742.279,A -85,B 0,C 180,E1 17111.873,E2 17111.873} C_VEL
LIN {X 0,Y 377.24,Z 731.002,A -85,B 0,C 180,E1 17108.382,E2 17108.382} C_VEL
LIN {X 0,Y 374.313,Z 725.995,A -85,B 0,C 180,E1 17106.749,E2 17106.749} C_VEL
LIN {X 0,Y 371.753,Z 721.506,A -85,B 0,C 180,E1 17105.246,E2 17105.246} C_VEL
LIN {X 0,Y 368.7,Z 716.322,A -85,B 0,C 180,E1 17103.42,E2 17103.42} C_VEL
LIN {X 0,Y 365.997,Z 711.606,A -85,B 0,C 180,E1 17101.722,E2 17101.722} C_VEL
LIN {X 0,Y 363.568,Z 707.42,A -85,B 0,C 180,E1 17100.157,E2 17100.157} C_VEL
LIN {X 0,Y 360.586,Z 702.71,A -85,B 0,C 180,E1 17098.252,E2 17098.252} C_VEL
LIN {X 0,Y 360.022,Z 701.316,A -85,B 0,C 180,E1 17097.771,E2 17097.771} C_VEL
LIN {X 0,Y 357.682,Z 698.097,A -85,B 0,C 180,E1 17096.313,E2 17096.313} C_VEL
LIN {X 0,Y 356.757,Z 695.876,A -85,B 0,C 180,E1 17095.499,E2 17095.499} C_VEL
LIN {X 0,Y 354.444,Z 692.776,A -85,B 0,C 180,E1 17094.009,E2 17094.009} C_VEL
LIN {X 0,Y 353.873,Z 690.652,A -85,B 0,C 180,E1 17093.266,E2 17093.266} C_VEL
LIN {X 0,Y 353.866,Z 690.651,A -85,B 0,C 180,E1 17088.922,E2 17088.922} C_VEL
LIN {X 0,Y 353.861,Z 690.653,A -85,B 0,C 180,E1 17084.765,E2 17084.765} C_VEL
LIN {X 0,Y 353.86,Z 690.637,A -85,B 0,C 180,E1 17080.687,E2 17080.687} C_VEL
LIN {X 0,Y 353.87,Z 690.637,A -85,B 0,C 180,E1 17076.522,E2 17076.522} C_VEL
LIN {X 0,Y 353.866,Z 690.659,A -85,B 0,C 180,E1 17073.785,E2 17073.785} C_VEL
LIN {X 0,Y 354.984,Z 693.804,A -85,B 0,C 180,E1 17073.033,E2 17073.033} C_VEL
LIN {X 0,Y 357.491,Z 696.351,A -85,B 0,C 180,E1 17071.973,E2 17071.973} C_VEL
LIN {X 0,Y 359.257,Z 700.037,A -85,B 0,C 180,E1 17071.035,E2 17071.035} C_VEL
LIN {X 0,Y 361.052,Z 702.169,A -85,B 0,C 180,E1 17070.284,E2 17070.284} C_VEL
LIN {X 0,Y 363.304,Z 706.175,A -85,B 0,C 180,E1 17069.209,E2 17069.209} C_VEL
LIN {X 0,Y 364.71,Z 708.413,A -85,B 0,C 180,E1 17068.608,E2 17068.608} C_VEL
LIN {X 0,Y 368.155,Z 714.241,A -85,B 0,C 180,E1 17067.1,E2 17067.1} C_VEL
LIN {X 0,Y 372.785,Z 722.274,A -85,B 0,C 180,E1 17065.157,E2 17065.157} C_VEL
LIN {X 0,Y 379.602,Z 735.404,A -85,B 0,C 180,E1 17062.332,E2 17062.332} C_VEL
LIN {X 0,Y 386.241,Z 749.435,A -85,B 0,C 180,E1 17059.671,E2 17059.671} C_VEL
LIN {X 0,Y 393.343,Z 766.409,A -85,B 0,C 180,E1 17056.847,E2 17056.847} C_VEL
LIN {X 0,Y 395.138,Z 771.497,A -85,B 0,C 180,E1 17056.105,E2 17056.105} C_VEL
LIN {X 0,Y 394.801,Z 779.344,A -85,B 0,C 180,E1 17055.548,E2 17055.548} C_VEL
LIN {X 0,Y 398.078,Z 808.112,A -85,B 0,C 180,E1 17054.34,E2 17054.34} C_VEL
LIN {X 0,Y 388.969,Z 1040.286,A -85,B 0,C 180,E1 17049.858,E2 17049.858} C_VEL
LIN {X 0,Y 387.491,Z 1060.983,A -85,B 0,C 180,E1 17049.21,E2 17049.21} C_VEL
LIN {X 0,Y 385.327,Z 1081.768,A -85,B 0,C 180,E1 17048.28,E2 17048.28} C_VEL
LIN {X 0,Y 382.682,Z 1101.267,A -85,B 0,C 180,E1 17047.123,E2 17047.123} C_VEL
LIN {X 0,Y 379.711,Z 1119.393,A -85,B 0,C 180,E1 17045.772,E2 17045.772} C_VEL
LIN {X 0,Y 376.26,Z 1137.53,A -85,B 0,C 180,E1 17044.103,E2 17044.103} C_VEL
LIN {X 0,Y 372.501,Z 1155.198,A -85,B 0,C 180,E1 17042.104,E2 17042.104} C_VEL
LIN {X 0,Y 368.808,Z 1171.054,A -85,B 0,C 180,E1 17039.922,E2 17039.922} C_VEL
LIN {X 0,Y 365.314,Z 1185.382,A -85,B 0,C 180,E1 17037.551,E2 17037.551} C_VEL
LIN {X 0,Y 362.11,Z 1198.301,A -85,B 0,C 180,E1 17034.989,E2 17034.989} C_VEL
LIN {X 0,Y 359.132,Z 1210.468,A -85,B 0,C 180,E1 17032.076,E2 17032.076} C_VEL
LIN {X 0,Y 356.792,Z 1220.539,A -85,B 0,C 180,E1 17029.139,E2 17029.139} C_VEL
LIN {X 0,Y 354.964,Z 1229.206,A -85,B 0,C 180,E1 17026.023,E2 17026.023} C_VEL
LIN {X 0,Y 354.378,Z 1232.205,A -85,B 0,C 180,E1 17024.751,E2 17024.751} C_VEL
LIN {X 0,Y 352.96,Z 1234.896,A -85,B 0,C 180,E1 17023.594,E2 17023.594} C_VEL
LIN {X 0,Y 345.853,Z 1241.142,A -85,B 0,C 180,E1 17020.467,E2 17020.467} C_VEL
LIN {X 0,Y 344.887,Z 1242.743,A -85,B 0,C 180,E1 17019.403,E2 17019.403} C_VEL
LIN {X 0,Y 344.458,Z 1246.341,A -85,B 0,C 180,E1 17015.997,E2 17015.997} C_VEL
LIN {X 0,Y 344.292,Z 1248.308,A -85,B 0,C 180,E1 17012.662,E2 17012.662} C_VEL
LIN {X 0,Y 344.257,Z 1248.788,A -85,B 0,C 180,E1 17009.334,E2 17009.334} C_VEL
LIN {X 0,Y 344.335,Z 1247.792,A -85,B 0,C 180,E1 17006.003,E2 17006.003} C_VEL
LIN {X 0,Y 344.582,Z 1245.222,A -85,B 0,C 180,E1 17002.664,E2 17002.664} C_VEL
LIN {X 0,Y 345.117,Z 1241.041,A -85,B 0,C 180,E1 16999.314,E2 16999.314} C_VEL
LIN {X 0,Y 346.113,Z 1235.185,A -85,B 0,C 180,E1 16995.956,E2 16995.956} C_VEL
LIN {X 0,Y 347.703,Z 1227.505,A -85,B 0,C 180,E1 16992.598,E2 16992.598} C_VEL
LIN {X 0,Y 349.858,Z 1218.321,A -85,B 0,C 180,E1 16989.419,E2 16989.419} C_VEL
LIN {X 0,Y 352.549,Z 1207.685,A -85,B 0,C 180,E1 16986.428,E2 16986.428} C_VEL
LIN {X 0,Y 355.709,Z 1195.607,A -85,B 0,C 180,E1 16983.632,E2 16983.632} C_VEL
LIN {X 0,Y 359.24,Z 1182.008,A -85,B 0,C 180,E1 16981.034,E2 16981.034} C_VEL
LIN {X 0,Y 362.923,Z 1167.409,A -85,B 0,C 180,E1 16978.713,E2 16978.713} C_VEL
LIN {X 0,Y 366.746,Z 1151.323,A -85,B 0,C 180,E1 16976.583,E2 16976.583} C_VEL
LIN {X 0,Y 370.615,Z 1133.485,A -85,B 0,C 180,E1 16974.641,E2 16974.641} C_VEL
LIN {X 0,Y 374.108,Z 1115.338,A -85,B 0,C 180,E1 16973.033,E2 16973.033} C_VEL
LIN {X 0,Y 377.079,Z 1097.428,A -85,B 0,C 180,E1 16971.746,E2 16971.746} C_VEL
LIN {X 0,Y 379.77,Z 1077.403,A -85,B 0,C 180,E1 16970.616,E2 16970.616} C_VEL
LIN {X 0,Y 381.813,Z 1057.012,A -85,B 0,C 180,E1 16969.765,E2 16969.765} C_VEL
LIN {X 0,Y 383.129,Z 1036.756,A -85,B 0,C 180,E1 16969.179,E2 16969.179} C_VEL
LIN {X 0,Y 391.918,Z 820.334,A -85,B 0,C 180,E1 16964.966,E2 16964.966} C_VEL
LIN {X 0,Y 384.444,Z 781.867,A -85,B 0,C 180,E1 16962.789,E2 16962.789} C_VEL
LIN {X 0,Y 384.385,Z 779.292,A -85,B 0,C 180,E1 16962.556,E2 16962.556} C_VEL
LIN {X 0,Y 384.518,Z 776.434,A -85,B 0,C 180,E1 16962.225,E2 16962.225} C_VEL
LIN {X 0,Y 383.851,Z 774.953,A -85,B 0,C 180,E1 16961.924,E2 16961.924} C_VEL
LIN {X 0,Y 381.123,Z 775.47,A -85,B 0,C 180,E1 16961.46,E2 16961.46} C_VEL
LIN {X 0,Y 375.73,Z 814.069,A -85,B 0,C 180,E1 16957.281,E2 16957.281} C_VEL
LIN {X 0,Y 370.493,Z 855.495,A -85,B 0,C 180,E1 16952.851,E2 16952.851} C_VEL
LIN {X 0,Y 368.917,Z 870.145,A -85,B 0,C 180,E1 16951.34,E2 16951.34} C_VEL
LIN {X 0,Y 369.868,Z 880.274,A -85,B 0,C 180,E1 16950.918,E2 16950.918} C_VEL
LIN {X 0,Y 361.074,Z 1037.813,A -85,B 0,C 180,E1 16946.539,E2 16946.539} C_VEL
LIN {X 0,Y 360.174,Z 1056.265,A -85,B 0,C 180,E1 16945.773,E2 16945.773} C_VEL
LIN {X 0,Y 358.846,Z 1073.954,A -85,B 0,C 180,E1 16944.722,E2 16944.722} C_VEL
LIN {X 0,Y 357.25,Z 1090.636,A -85,B 0,C 180,E1 16943.418,E2 16943.418} C_VEL
LIN {X 0,Y 355.493,Z 1106.141,A -85,B 0,C 180,E1 16941.881,E2 16941.881} C_VEL
LIN {X 0,Y 353.575,Z 1121.19,A -85,B 0,C 180,E1 16940.01,E2 16940.01} C_VEL
LIN {X 0,Y 351.759,Z 1134.588,A -85,B 0,C 180,E1 16937.964,E2 16937.964} C_VEL
LIN {X 0,Y 350.116,Z 1146.418,A -85,B 0,C 180,E1 16935.742,E2 16935.742} C_VEL
LIN {X 0,Y 348.646,Z 1157.117,A -85,B 0,C 180,E1 16933.264,E2 16933.264} C_VEL
LIN {X 0,Y 347.506,Z 1166.304,A -85,B 0,C 180,E1 16930.612,E2 16930.612} C_VEL
LIN {X 0,Y 346.714,Z 1173.804,A -85,B 0,C 180,E1 16927.79,E2 16927.79} C_VEL
LIN {X 0,Y 346.264,Z 1179.413,A -85,B 0,C 180,E1 16924.97,E2 16924.97} C_VEL
LIN {X 0,Y 346.109,Z 1183.271,A -85,B 0,C 180,E1 16922.153,E2 16922.153} C_VEL
LIN {X 0,Y 346.186,Z 1185.488,A -85,B 0,C 180,E1 16919.173,E2 16919.173} C_VEL
LIN {X 0,Y 346.5,Z 1185.971,A -85,B 0,C 180,E1 16916.195,E2 16916.195} C_VEL
LIN {X 0,Y 347.078,Z 1184.738,A -85,B 0,C 180,E1 16913.383,E2 16913.383} C_VEL
LIN {X 0,Y 348.037,Z 1181.662,A -85,B 0,C 180,E1 16910.409,E2 16910.409} C_VEL
LIN {X 0,Y 349.369,Z 1177.028,A -85,B 0,C 180,E1 16907.606,E2 16907.606} C_VEL
LIN {X 0,Y 351.168,Z 1170.437,A -85,B 0,C 180,E1 16904.815,E2 16904.815} C_VEL
LIN {X 0,Y 353.226,Z 1162.921,A -85,B 0,C 180,E1 16902.37,E2 16902.37} C_VEL
LIN {X 0,Y 355.681,Z 1153.329,A -85,B 0,C 180,E1 16899.943,E2 16899.943} C_VEL
LIN {X 0,Y 358.374,Z 1142.316,A -85,B 0,C 180,E1 16897.702,E2 16897.702} C_VEL
LIN {X 0,Y 361.272,Z 1129.201,A -85,B 0,C 180,E1 16895.581,E2 16895.581} C_VEL
LIN {X 0,Y 363.912,Z 1115.745,A -85,B 0,C 180,E1 16893.834,E2 16893.834} C_VEL
LIN {X 0,Y 366.47,Z 1100.87,A -85,B 0,C 180,E1 16892.278,E2 16892.278} C_VEL
LIN {X 0,Y 368.867,Z 1083.902,A -85,B 0,C 180,E1 16890.886,E2 16890.886} C_VEL
LIN {X 0,Y 372.183,Z 1058.443,A -85,B 0,C 180,E1 16889.308,E2 16889.308} C_VEL
LIN {X 0,Y 378.138,Z 1029.933,A -85,B 0,C 180,E1 16887.716,E2 16887.716} C_VEL
LIN {X 0,Y 392.277,Z 974.412,A -85,B 0,C 180,E1 16885.073,E2 16885.073} C_VEL
LIN {X 0,Y 401.286,Z 937.757,A -85,B 0,C 180,E1 16883.591,E2 16883.591} C_VEL
LIN {X 0,Y 412.018,Z 922.445,A -85,B 0,C 180,E1 16882.747,E2 16882.747} C_VEL
LIN {X 0,Y 415.081,Z 918.33,A -85,B 0,C 180,E1 16882.452,E2 16882.452} C_VEL
LIN {X 0,Y 414.609,Z 925.972,A -85,B 0,C 180,E1 16880.458,E2 16880.458} C_VEL
LIN {X 0,Y 416.64,Z 934.008,A -85,B 0,C 180,E1 16878.482,E2 16878.482} C_VEL
LIN {X 0,Y 417.17,Z 935.4,A -85,B 0,C 180,E1 16878.168,E2 16878.168} C_VEL
LIN {X 0,Y 407.765,Z 954.035,A -85,B 0,C 180,E1 16877.498,E2 16877.498} C_VEL
LIN {X 0,Y 400.712,Z 968.648,A -85,B 0,C 180,E1 16876.992,E2 16876.992} C_VEL
LIN {X 0,Y 395.628,Z 994.265,A -85,B 0,C 180,E1 16876.588,E2 16876.588} C_VEL
LIN {X 0,Y 389.939,Z 1020.766,A -85,B 0,C 180,E1 16876.145,E2 16876.145} C_VEL
LIN {X 0,Y 386.824,Z 1036.948,A -85,B 0,C 180,E1 16875.605,E2 16875.605} C_VEL
LIN {X 0,Y 381.25,Z 1067.04,A -85,B 0,C 180,E1 16874.236,E2 16874.236} C_VEL
LIN {X 0,Y 376.004,Z 1094.153,A -85,B 0,C 180,E1 16872.695,E2 16872.695} C_VEL
LIN {X 0,Y 371.077,Z 1119.59,A -85,B 0,C 180,E1 16870.902,E2 16870.902} C_VEL
LIN {X 0,Y 368.059,Z 1136.277,A -85,B 0,C 180,E1 16869.562,E2 16869.562} C_VEL
LIN {X 0,Y 365.828,Z 1155.88,A -85,B 0,C 180,E1 16868.148,E2 16868.148} C_VEL
LIN {X 0,Y 363.229,Z 1174.727,A -85,B 0,C 180,E1 16866.484,E2 16866.484} C_VEL
LIN {X 0,Y 360.357,Z 1192.692,A -85,B 0,C 180,E1 16864.571,E2 16864.571} C_VEL
LIN {X 0,Y 357.278,Z 1210.286,A -85,B 0,C 180,E1 16862.312,E2 16862.312} C_VEL
LIN {X 0,Y 354.464,Z 1225.681,A -85,B 0,C 180,E1 16859.953,E2 16859.953} C_VEL
LIN {X 0,Y 351.855,Z 1239.769,A -85,B 0,C 180,E1 16857.41,E2 16857.41} C_VEL
LIN {X 0,Y 349.472,Z 1253.322,A -85,B 0,C 180,E1 16854.511,E2 16854.511} C_VEL
LIN {X 0,Y 347.62,Z 1264.75,A -85,B 0,C 180,E1 16851.603,E2 16851.603} C_VEL
LIN {X 0,Y 346.185,Z 1274.848,A -85,B 0,C 180,E1 16848.525,E2 16848.525} C_VEL
LIN {X 0,Y 345.163,Z 1283.46,A -85,B 0,C 180,E1 16845.285,E2 16845.285} C_VEL
LIN {X 0,Y 344.615,Z 1290.264,A -85,B 0,C 180,E1 16842.059,E2 16842.059} C_VEL
LIN {X 0,Y 344.352,Z 1295.623,A -85,B 0,C 180,E1 16838.685,E2 16838.685} C_VEL
LIN {X 0,Y 344.311,Z 1299.104,A -85,B 0,C 180,E1 16835.5,E2 16835.5} C_VEL
LIN {X 0,Y 344.338,Z 1300.965,A -85,B 0,C 180,E1 16832.331,E2 16832.331} C_VEL
LIN {X 0,Y 344.341,Z 1301.307,A -85,B 0,C 180,E1 16829.169,E2 16829.169} C_VEL
LIN {X 0,Y 344.317,Z 1300.181,A -85,B 0,C 180,E1 16826.004,E2 16826.004} C_VEL
LIN {X 0,Y 344.293,Z 1297.466,A -85,B 0,C 180,E1 16822.827,E2 16822.827} C_VEL
LIN {X 0,Y 344.414,Z 1293.168,A -85,B 0,C 180,E1 16819.632,E2 16819.632} C_VEL
LIN {X 0,Y 344.777,Z 1286.889,A -85,B 0,C 180,E1 16816.244,E2 16816.244} C_VEL
LIN {X 0,Y 345.534,Z 1279.145,A -85,B 0,C 180,E1 16813.008,E2 16813.008} C_VEL
LIN {X 0,Y 346.738,Z 1269.477,A -85,B 0,C 180,E1 16809.756,E2 16809.756} C_VEL
LIN {X 0,Y 348.403,Z 1258.263,A -85,B 0,C 180,E1 16806.67,E2 16806.67} C_VEL
LIN {X 0,Y 350.521,Z 1245.609,A -85,B 0,C 180,E1 16803.761,E2 16803.761} C_VEL
LIN {X 0,Y 353.002,Z 1231.538,A -85,B 0,C 180,E1 16801.031,E2 16801.031} C_VEL
LIN {X 0,Y 356.747,Z 1212.975,A -85,B 0,C 180,E1 16797.823,E2 16797.823} C_VEL
LIN {X 0,Y 360.393,Z 1195.631,A -85,B 0,C 180,E1 16795.288,E2 16795.288} C_VEL
LIN {X 0,Y 364.204,Z 1177.266,A -85,B 0,C 180,E1 16793.024,E2 16793.024} C_VEL
LIN {X 0,Y 368.274,Z 1157.236,A -85,B 0,C 180,E1 16790.939,E2 16790.939} C_VEL
LIN {X 0,Y 372.263,Z 1136.82,A -85,B 0,C 180,E1 16789.156,E2 16789.156} C_VEL
LIN {X 0,Y 376.327,Z 1114.28,A -85,B 0,C 180,E1 16787.559,E2 16787.559} C_VEL
LIN {X 0,Y 380.035,Z 1091.442,A -85,B 0,C 180,E1 16786.269,E2 16786.269} C_VEL
LIN {X 0,Y 383.269,Z 1068.278,A -85,B 0,C 180,E1 16785.268,E2 16785.268} C_VEL
LIN {X 0,Y 385.79,Z 1043.904,A -85,B 0,C 180,E1 16784.491,E2 16784.491} C_VEL
LIN {X 0,Y 387.658,Z 1021.114,A -85,B 0,C 180,E1 16783.973,E2 16783.973} C_VEL
LIN {X 0,Y 389.987,Z 1004.934,A -85,B 0,C 180,E1 16783.699,E2 16783.699} C_VEL
LIN {X 0,Y 403.094,Z 974.211,A -85,B 0,C 180,E1 16782.237,E2 16782.237} C_VEL
LIN {X 0,Y 413.377,Z 954.145,A -85,B 0,C 180,E1 16781.509,E2 16781.509} C_VEL
LIN {X 0,Y 421.013,Z 938.826,A -85,B 0,C 180,E1 16780.955,E2 16780.955} C_VEL
LIN {X 0,Y 413.232,Z 923.474,A -85,B 0,C 180,E1 16778.627,E2 16778.627} C_VEL
LIN {X 0,Y 407.734,Z 907.537,A -85,B 0,C 180,E1 16776.401,E2 16776.401} C_VEL
LIN {X 0,Y 404.07,Z 889.515,A -85,B 0,C 180,E1 16774.088,E2 16774.088} C_VEL
LIN {X 0,Y 402.52,Z 870.317,A -85,B 0,C 180,E1 16771.842,E2 16771.842} C_VEL
LIN {X 0,Y 402.986,Z 849.92,A -85,B 0,C 180,E1 16769.677,E2 16769.677} C_VEL
LIN {X 0,Y 405.755,Z 826.411,A -85,B 0,C 180,E1 16767.439,E2 16767.439} C_VEL
LIN {X 0,Y 409.372,Z 805.589,A -85,B 0,C 180,E1 16765.614,E2 16765.614} C_VEL
LIN {X 0,Y 400.724,Z 788.566,A -85,B 0,C 180,E1 16761.979,E2 16761.979} C_VEL
LIN {X 0,Y 391.818,Z 771.736,A -85,B 0,C 180,E1 16757.985,E2 16757.985} C_VEL
LIN {X 0,Y 383.882,Z 757.28,A -85,B 0,C 180,E1 16754.172,E2 16754.172} C_VEL
LIN {X 0,Y 376.031,Z 743.292,A -85,B 0,C 180,E1 16750.107,E2 16750.107} C_VEL
LIN {X 0,Y 369.767,Z 732.622,A -85,B 0,C 180,E1 16746.677,E2 16746.677} C_VEL
LIN {X 0,Y 366.614,Z 727.277,A -85,B 0,C 180,E1 16744.85,E2 16744.85} C_VEL
LIN {X 0,Y 364.104,Z 722.838,A -85,B 0,C 180,E1 16743.306,E2 16743.306} C_VEL
LIN {X 0,Y 361.051,Z 717.686,A -85,B 0,C 180,E1 16741.406,E2 16741.406} C_VEL
LIN {X 0,Y 357.962,Z 712.461,A -85,B 0,C 180,E1 16739.401,E2 16739.401} C_VEL
LIN {X 0,Y 355.595,Z 708.212,A -85,B 0,C 180,E1 16737.744,E2 16737.744} C_VEL
LIN {X 0,Y 352.836,Z 704.011,A -85,B 0,C 180,E1 16735.924,E2 16735.924} C_VEL
LIN {X 0,Y 352.051,Z 702.284,A -85,B 0,C 180,E1 16735.275,E2 16735.275} C_VEL
LIN {X 0,Y 349.795,Z 699.115,A -85,B 0,C 180,E1 16733.764,E2 16733.764} C_VEL
LIN {X 0,Y 348.847,Z 696.88,A -85,B 0,C 180,E1 16732.92,E2 16732.92} C_VEL
LIN {X 0,Y 346.566,Z 693.937,A -85,B 0,C 180,E1 16731.371,E2 16731.371} C_VEL
LIN {X 0,Y 345.932,Z 691.645,A -85,B 0,C 180,E1 16730.517,E2 16730.517} C_VEL
LIN {X 0,Y 345.924,Z 691.641,A -85,B 0,C 180,E1 16726.119,E2 16726.119} C_VEL
LIN {X 0,Y 345.924,Z 691.634,A -85,B 0,C 180,E1 16721.975,E2 16721.975} C_VEL
LIN {X 0,Y 345.927,Z 691.633,A -85,B 0,C 180,E1 16717.75,E2 16717.75} C_VEL
LIN {X 0,Y 345.954,Z 691.826,A -85,B 0,C 180,E1 16716.178,E2 16716.178} C_VEL
LIN {X 0,Y 347.16,Z 695.016,A -85,B 0,C 180,E1 16715.315,E2 16715.315} C_VEL
LIN {X 0,Y 349.847,Z 697.83,A -85,B 0,C 180,E1 16714.07,E2 16714.07} C_VEL
LIN {X 0,Y 351.546,Z 701.186,A -85,B 0,C 180,E1 16713.113,E2 16713.113} C_VEL
LIN {X 0,Y 353.546,Z 703.605,A -85,B 0,C 180,E1 16712.184,E2 16712.184} C_VEL
LIN {X 0,Y 355.726,Z 707.362,A -85,B 0,C 180,E1 16711.089,E2 16711.089} C_VEL
LIN {X 0,Y 357.109,Z 709.33,A -85,B 0,C 180,E1 16710.476,E2 16710.476} C_VEL
LIN {X 0,Y 360.376,Z 714.844,A -85,B 0,C 180,E1 16708.932,E2 16708.932} C_VEL
LIN {X 0,Y 365.538,Z 723.584,A -85,B 0,C 180,E1 16706.647,E2 16706.647} C_VEL
LIN {X 0,Y 372.519,Z 736.861,A -85,B 0,C 180,E1 16703.617,E2 16703.617} C_VEL
LIN {X 0,Y 379.3,Z 750.912,A -85,B 0,C 180,E1 16700.804,E2 16700.804} C_VEL
LIN {X 0,Y 386.34,Z 767.542,A -85,B 0,C 180,E1 16697.909,E2 16697.909} C_VEL
LIN {X 0,Y 389.268,Z 774.971,A -85,B 0,C 180,E1 16696.751,E2 16696.751} C_VEL
LIN {X 0,Y 389.131,Z 780.127,A -85,B 0,C 180,E1 16696.398,E2 16696.398} C_VEL
LIN {X 0,Y 392.368,Z 809.514,A -85,B 0,C 180,E1 16695.137,E2 16695.137} C_VEL
LIN {X 0,Y 382.87,Z 1040.903,A -85,B 0,C 180,E1 16690.622,E2 16690.622} C_VEL
LIN {X 0,Y 381.34,Z 1061.541,A -85,B 0,C 180,E1 16689.968,E2 16689.968} C_VEL
LIN {X 0,Y 379.088,Z 1082.345,A -85,B 0,C 180,E1 16689.028,E2 16689.028} C_VEL
LIN {X 0,Y 376.337,Z 1101.855,A -85,B 0,C 180,E1 16687.858,E2 16687.858} C_VEL
LIN {X 0,Y 373.243,Z 1119.989,A -85,B 0,C 180,E1 16686.49,E2 16686.49} C_VEL
LIN {X 0,Y 369.641,Z 1138.131,A -85,B 0,C 180,E1 16684.801,E2 16684.801} C_VEL
LIN {X 0,Y 365.715,Z 1155.803,A -85,B 0,C 180,E1 16682.773,E2 16682.773} C_VEL
LIN {X 0,Y 361.846,Z 1171.663,A -85,B 0,C 180,E1 16680.558,E2 16680.558} C_VEL
LIN {X 0,Y 358.18,Z 1185.993,A -85,B 0,C 180,E1 16678.148,E2 16678.148} C_VEL
LIN {X 0,Y 354.798,Z 1198.915,A -85,B 0,C 180,E1 16675.541,E2 16675.541} C_VEL
LIN {X 0,Y 351.646,Z 1211.084,A -85,B 0,C 180,E1 16672.572,E2 16672.572} C_VEL
LIN {X 0,Y 349.16,Z 1221.155,A -85,B 0,C 180,E1 16669.574,E2 16669.574} C_VEL
LIN {X 0,Y 347.205,Z 1229.822,A -85,B 0,C 180,E1 16666.392,E2 16666.392} C_VEL
LIN {X 0,Y 345.78,Z 1237.12,A -85,B 0,C 180,E1 16662.973,E2 16662.973} C_VEL
LIN {X 0,Y 344.907,Z 1242.594,A -85,B 0,C 180,E1 16659.51,E2 16659.51} C_VEL
LIN {X 0,Y 344.887,Z 1242.743,A -85,B 0,C 180,E1 16659.403,E2 16659.403} C_VEL
LIN {X 0,Y 343.696,Z 1244.449,A -85,B 0,C 180,E1 16658.158,E2 16658.158} C_VEL
LIN {X 0,Y 338.846,Z 1247.172,A -85,B 0,C 180,E1 16655.794,E2 16655.794} C_VEL
LIN {X 0,Y 336.519,Z 1248.356,A -85,B 0,C 180,E1 16654.142,E2 16654.142} C_VEL
LIN {X 0,Y 336.352,Z 1248.564,A -85,B 0,C 180,E1 16653.669,E2 16653.669} C_VEL
LIN {X 0,Y 336.284,Z 1249.428,A -85,B 0,C 180,E1 16650.34,E2 16650.34} C_VEL
LIN {X 0,Y 336.324,Z 1248.827,A -85,B 0,C 180,E1 16646.932,E2 16646.932} C_VEL
LIN {X 0,Y 336.541,Z 1246.586,A -85,B 0,C 180,E1 16643.346,E2 16643.346} C_VEL
LIN {X 0,Y 337.036,Z 1242.86,A -85,B 0,C 180,E1 16639.919,E2 16639.919} C_VEL
LIN {X 0,Y 337.981,Z 1237.482,A -85,B 0,C 180,E1 16636.484,E2 16636.484} C_VEL
LIN {X 0,Y 339.508,Z 1230.266,A -85,B 0,C 180,E1 16633.048,E2 16633.048} C_VEL
LIN {X 0,Y 341.62,Z 1221.552,A -85,B 0,C 180,E1 16629.795,E2 16629.795} C_VEL
LIN {X 0,Y 344.279,Z 1211.426,A -85,B 0,C 180,E1 16626.735,E2 16626.735} C_VEL
LIN {X 0,Y 347.635,Z 1199.191,A -85,B 0,C 180,E1 16623.708,E2 16623.708} C_VEL
LIN {X 0,Y 351.46,Z 1185.3,A -85,B 0,C 180,E1 16620.89,E2 16620.89} C_VEL
LIN {X 0,Y 355.359,Z 1170.7,A -85,B 0,C 180,E1 16618.443,E2 16618.443} C_VEL
LIN {X 0,Y 359.301,Z 1155.158,A -85,B 0,C 180,E1 16616.277,E2 16616.277} C_VEL
LIN {X 0,Y 363.275,Z 1138.013,A -85,B 0,C 180,E1 16614.302,E2 16614.302} C_VEL
LIN {X 0,Y 367.048,Z 1119.76,A -85,B 0,C 180,E1 16612.593,E2 16612.593} C_VEL
LIN {X 0,Y 370.279,Z 1101.404,A -85,B 0,C 180,E1 16611.209,E2 16611.209} C_VEL
LIN {X 0,Y 373.07,Z 1082.117,A -85,B 0,C 180,E1 16610.057,E2 16610.057} C_VEL
LIN {X 0,Y 375.354,Z 1061.609,A -85,B 0,C 180,E1 16609.131,E2 16609.131} C_VEL
LIN {X 0,Y 376.951,Z 1040.407,A -85,B 0,C 180,E1 16608.464,E2 16608.464} C_VEL
LIN {X 0,Y 386.269,Z 822.151,A -85,B 0,C 180,E1 16604.157,E2 16604.157} C_VEL
LIN {X 0,Y 379.115,Z 784.36,A -85,B 0,C 180,E1 16601.97,E2 16601.97} C_VEL
LIN {X 0,Y 375.513,Z 787.176,A -85,B 0,C 180,E1 16601.428,E2 16601.428} C_VEL
LIN {X 0,Y 373.28,Z 787.45,A -85,B 0,C 180,E1 16601.04,E2 16601.04} C_VEL
LIN {X 0,Y 367.758,Z 825.891,A -85,B 0,C 180,E1 16596.834,E2 16596.834} C_VEL
LIN {X 0,Y 362.454,Z 867.539,A -85,B 0,C 180,E1 16592.355,E2 16592.355} C_VEL
LIN {X 0,Y 362.15,Z 871.36,A -85,B 0,C 180,E1 16591.989,E2 16591.989} C_VEL
LIN {X 0,Y 363.039,Z 881.326,A -85,B 0,C 180,E1 16591.559,E2 16591.559} C_VEL
LIN {X 0,Y 353.812,Z 1038.083,A -85,B 0,C 180,E1 16587.076,E2 16587.076} C_VEL
LIN {X 0,Y 352.857,Z 1056.833,A -85,B 0,C 180,E1 16586.286,E2 16586.286} C_VEL
LIN {X 0,Y 351.508,Z 1074.28,A -85,B 0,C 180,E1 16585.237,E2 16585.237} C_VEL
LIN {X 0,Y 349.777,Z 1091.702,A -85,B 0,C 180,E1 16583.85,E2 16583.85} C_VEL
LIN {X 0,Y 347.962,Z 1107.132,A -85,B 0,C 180,E1 16582.291,E2 16582.291} C_VEL
LIN {X 0,Y 346.053,Z 1121.622,A -85,B 0,C 180,E1 16580.464,E2 16580.464} C_VEL
LIN {X 0,Y 344.084,Z 1135.66,A -85,B 0,C 180,E1 16578.291,E2 16578.291} C_VEL
LIN {X 0,Y 342.437,Z 1147.171,A -85,B 0,C 180,E1 16576.105,E2 16576.105} C_VEL
LIN {X 0,Y 340.895,Z 1157.983,A -85,B 0,C 180,E1 16573.571,E2 16573.571} C_VEL
LIN {X 0,Y 339.692,Z 1167.285,A -85,B 0,C 180,E1 16570.859,E2 16570.859} C_VEL
LIN {X 0,Y 338.902,Z 1174.542,A -85,B 0,C 180,E1 16568.142,E2 16568.142} C_VEL
LIN {X 0,Y 338.4,Z 1180.343,A -85,B 0,C 180,E1 16565.256,E2 16565.256} C_VEL
LIN {X 0,Y 338.225,Z 1184.592,A -85,B 0,C 180,E1 16562.203,E2 16562.203} C_VEL
LIN {X 0,Y 338.302,Z 1186.844,A -85,B 0,C 180,E1 16559.323,E2 16559.323} C_VEL
LIN {X 0,Y 338.633,Z 1187.508,A -85,B 0,C 180,E1 16556.276,E2 16556.276} C_VEL
LIN {X 0,Y 339.283,Z 1186.435,A -85,B 0,C 180,E1 16553.284,E2 16553.284} C_VEL
LIN {X 0,Y 340.341,Z 1183.449,A -85,B 0,C 180,E1 16550.19,E2 16550.19} C_VEL
LIN {X 0,Y 341.78,Z 1178.943,A -85,B 0,C 180,E1 16547.326,E2 16547.326} C_VEL
LIN {X 0,Y 343.721,Z 1172.535,A -85,B 0,C 180,E1 16544.478,E2 16544.478} C_VEL
LIN {X 0,Y 346.082,Z 1164.62,A -85,B 0,C 180,E1 16541.819,E2 16541.819} C_VEL
LIN {X 0,Y 348.74,Z 1155.145,A -85,B 0,C 180,E1 16539.351,E2 16539.351} C_VEL
LIN {X 0,Y 351.637,Z 1144.262,A -85,B 0,C 180,E1 16537.074,E2 16537.074} C_VEL
LIN {X 0,Y 354.919,Z 1130.736,A -85,B 0,C 180,E1 16534.825,E2 16534.825} C_VEL
LIN {X 0,Y 358.155,Z 1115.634,A -85,B 0,C 180,E1 16532.843,E2 16532.843} C_VEL
LIN {X 0,Y 361.243,Z 1098.945,A -85,B 0,C 180,E1 16531.12,E2 16531.12} C_VEL
LIN {X 0,Y 363.935,Z 1081.537,A -85,B 0,C 180,E1 16529.726,E2 16529.726} C_VEL
LIN {X 0,Y 367.78,Z 1058.971,A -85,B 0,C 180,E1 16528.261,E2 16528.261} C_VEL
LIN {X 0,Y 374.657,Z 1031.617,A -85,B 0,C 180,E1 16526.65,E2 16526.65} C_VEL
LIN {X 0,Y 388.249,Z 984.257,A -85,B 0,C 180,E1 16524.317,E2 16524.317} C_VEL
LIN {X 0,Y 399.288,Z 942.648,A -85,B 0,C 180,E1 16522.61,E2 16522.61} C_VEL
LIN {X 0,Y 409.879,Z 927.988,A -85,B 0,C 180,E1 16521.869,E2 16521.869} C_VEL
LIN {X 0,Y 410.344,Z 935.797,A -85,B 0,C 180,E1 16519.782,E2 16519.782} C_VEL
LIN {X 0,Y 411.133,Z 939.057,A -85,B 0,C 180,E1 16518.989,E2 16518.989} C_VEL
LIN {X 0,Y 403.461,Z 953.927,A -85,B 0,C 180,E1 16518.454,E2 16518.454} C_VEL
LIN {X 0,Y 398.566,Z 963.914,A -85,B 0,C 180,E1 16518.129,E2 16518.129} C_VEL
LIN {X 0,Y 392.164,Z 994.198,A -85,B 0,C 180,E1 16517.637,E2 16517.637} C_VEL
LIN {X 0,Y 385.953,Z 1020.563,A -85,B 0,C 180,E1 16517.172,E2 16517.172} C_VEL
LIN {X 0,Y 382.437,Z 1036.595,A -85,B 0,C 180,E1 16516.621,E2 16516.621} C_VEL
LIN {X 0,Y 375.669,Z 1068.923,A -85,B 0,C 180,E1 16515.071,E2 16515.071} C_VEL
LIN {X 0,Y 369.669,Z 1096.555,A -85,B 0,C 180,E1 16513.394,E2 16513.394} C_VEL
LIN {X 0,Y 364.138,Z 1122.777,A -85,B 0,C 180,E1 16511.434,E2 16511.434} C_VEL
LIN {X 0,Y 361.908,Z 1134.241,A -85,B 0,C 180,E1 16510.485,E2 16510.485} C_VEL
LIN {X 0,Y 359.667,Z 1153.253,A -85,B 0,C 180,E1 16509.128,E2 16509.128} C_VEL
LIN {X 0,Y 356.887,Z 1172.444,A -85,B 0,C 180,E1 16507.442,E2 16507.442} C_VEL
LIN {X 0,Y 353.81,Z 1190.435,A -85,B 0,C 180,E1 16505.524,E2 16505.524} C_VEL
LIN {X 0,Y 350.692,Z 1207.433,A -85,B 0,C 180,E1 16503.346,E2 16503.346} C_VEL
LIN {X 0,Y 347.545,Z 1223.498,A -85,B 0,C 180,E1 16500.9,E2 16500.9} C_VEL
LIN {X 0,Y 344.49,Z 1239.014,A -85,B 0,C 180,E1 16498.075,E2 16498.075} C_VEL
LIN {X 0,Y 341.911,Z 1252.693,A -85,B 0,C 180,E1 16495.09,E2 16495.09} C_VEL
LIN {X 0,Y 339.883,Z 1264.25,A -85,B 0,C 180,E1 16492.081,E2 16492.081} C_VEL
LIN {X 0,Y 338.285,Z 1274.712,A -85,B 0,C 180,E1 16488.795,E2 16488.795} C_VEL
LIN {X 0,Y 337.204,Z 1283.257,A -85,B 0,C 180,E1 16485.478,E2 16485.478} C_VEL
LIN {X 0,Y 336.631,Z 1289.962,A -85,B 0,C 180,E1 16482.175,E2 16482.175} C_VEL
LIN {X 0,Y 336.361,Z 1295.226,A -85,B 0,C 180,E1 16478.72,E2 16478.72} C_VEL
LIN {X 0,Y 336.328,Z 1298.613,A -85,B 0,C 180,E1 16475.46,E2 16475.46} C_VEL
LIN {X 0,Y 336.358,Z 1300.355,A -85,B 0,C 180,E1 16472.386,E2 16472.386} C_VEL
LIN {X 0,Y 336.364,Z 1300.698,A -85,B 0,C 180,E1 16469.149,E2 16469.149} C_VEL
LIN {X 0,Y 336.334,Z 1299.688,A -85,B 0,C 180,E1 16466.08,E2 16466.08} C_VEL
LIN {X 0,Y 336.305,Z 1297.021,A -85,B 0,C 180,E1 16462.828,E2 16462.828} C_VEL
LIN {X 0,Y 336.422,Z 1292.816,A -85,B 0,C 180,E1 16459.556,E2 16459.556} C_VEL
LIN {X 0,Y 336.771,Z 1287.003,A -85,B 0,C 180,E1 16456.261,E2 16456.261} C_VEL
LIN {X 0,Y 337.546,Z 1279.446,A -85,B 0,C 180,E1 16452.948,E2 16452.948} C_VEL
LIN {X 0,Y 338.791,Z 1269.926,A -85,B 0,C 180,E1 16449.621,E2 16449.621} C_VEL
LIN {X 0,Y 340.528,Z 1258.945,A -85,B 0,C 180,E1 16446.465,E2 16446.465} C_VEL
LIN {X 0,Y 342.744,Z 1246.563,A -85,B 0,C 180,E1 16443.492,E2 16443.492} C_VEL
LIN {X 0,Y 345.461,Z 1232.18,A -85,B 0,C 180,E1 16440.595,E2 16440.595} C_VEL
LIN {X 0,Y 348.356,Z 1217.046,A -85,B 0,C 180,E1 16438.026,E2 16438.026} C_VEL
LIN {X 0,Y 353.603,Z 1192.072,A -85,B 0,C 180,E1 16434.375,E2 16434.375} C_VEL
LIN {X 0,Y 357.81,Z 1172.669,A -85,B 0,C 180,E1 16432,E2 16432} C_VEL
LIN {X 0,Y 362.01,Z 1152.471,A -85,B 0,C 180,E1 16429.945,E2 16429.945} C_VEL
LIN {X 0,Y 366.466,Z 1130.093,A -85,B 0,C 180,E1 16428.053,E2 16428.053} C_VEL
LIN {X 0,Y 370.557,Z 1107.748,A -85,B 0,C 180,E1 16426.525,E2 16426.525} C_VEL
LIN {X 0,Y 374.328,Z 1084.422,A -85,B 0,C 180,E1 16425.276,E2 16425.276} C_VEL
LIN {X 0,Y 377.671,Z 1060.353,A -85,B 0,C 180,E1 16424.299,E2 16424.299} C_VEL
LIN {X 0,Y 379.836,Z 1037.117,A -85,B 0,C 180,E1 16423.605,E2 16423.605} C_VEL
LIN {X 0,Y 381.791,Z 1017.044,A -85,B 0,C 180,E1 16423.183,E2 16423.183} C_VEL
LIN {X 0,Y 383.676,Z 1004.24,A -85,B 0,C 180,E1 16422.978,E2 16422.978} C_VEL
LIN {X 0,Y 397.099,Z 973.214,A -85,B 0,C 180,E1 16421.491,E2 16421.491} C_VEL
LIN {X 0,Y 407.262,Z 953.47,A -85,B 0,C 180,E1 16420.771,E2 16420.771} C_VEL
LIN {X 0,Y 413.456,Z 941.247,A -85,B 0,C 180,E1 16420.328,E2 16420.328} C_VEL
LIN {X 0,Y 406.096,Z 925.743,A -85,B 0,C 180,E1 16417.99,E2 16417.99} C_VEL
LIN {X 0,Y 400.73,Z 908.863,A -85,B 0,C 180,E1 16415.633,E2 16415.633} C_VEL
LIN {X 0,Y 397.418,Z 890.321,A -85,B 0,C 180,E1 16413.261,E2 16413.261} C_VEL
LIN {X 0,Y 396.269,Z 870.806,A -85,B 0,C 180,E1 16410.979,E2 16410.979} C_VEL
LIN {X 0,Y 397.172,Z 849.66,A -85,B 0,C 180,E1 16408.739,E2 16408.739} C_VEL
LIN {X 0,Y 400.337,Z 825.798,A -85,B 0,C 180,E1 16406.483,E2 16406.483} C_VEL
LIN {X 0,Y 403.306,Z 809.895,A -85,B 0,C 180,E1 16405.083,E2 16405.083} C_VEL
LIN {X 0,Y 394.67,Z 792.875,A -85,B 0,C 180,E1 16401.396,E2 16401.396} C_VEL
LIN {X 0,Y 386.088,Z 776.643,A -85,B 0,C 180,E1 16397.482,E2 16397.482} C_VEL
LIN {X 0,Y 378.745,Z 763.154,A -85,B 0,C 180,E1 16393.9,E2 16393.9} C_VEL
LIN {X 0,Y 371.186,Z 749.549,A -85,B 0,C 180,E1 16389.927,E2 16389.927} C_VEL
LIN {X 0,Y 364.647,Z 738.409,A -85,B 0,C 180,E1 16386.296,E2 16386.296} C_VEL
LIN {X 0,Y 361.489,Z 733.018,A -85,B 0,C 180,E1 16384.441,E2 16384.441} C_VEL
LIN {X 0,Y 358.939,Z 728.584,A -85,B 0,C 180,E1 16382.874,E2 16382.874} C_VEL
LIN {X 0,Y 356,Z 723.595,A -85,B 0,C 180,E1 16381.024,E2 16381.024} C_VEL
LIN {X 0,Y 353.229,Z 718.79,A -85,B 0,C 180,E1 16379.189,E2 16379.189} C_VEL
LIN {X 0,Y 350.077,Z 713.527,A -85,B 0,C 180,E1 16377.053,E2 16377.053} C_VEL
LIN {X 0,Y 347.793,Z 709.459,A -85,B 0,C 180,E1 16375.383,E2 16375.383} C_VEL
LIN {X 0,Y 344.911,Z 704.962,A -85,B 0,C 180,E1 16373.341,E2 16373.341} C_VEL
LIN {X 0,Y 344.098,Z 703.257,A -85,B 0,C 180,E1 16372.654,E2 16372.654} C_VEL
LIN {X 0,Y 341.673,Z 699.715,A -85,B 0,C 180,E1 16370.907,E2 16370.907} C_VEL
LIN {X 0,Y 340.941,Z 697.897,A -85,B 0,C 180,E1 16370.18,E2 16370.18} C_VEL
LIN {X 0,Y 338.664,Z 694.999,A -85,B 0,C 180,E1 16368.569,E2 16368.569} C_VEL
LIN {X 0,Y 337.991,Z 692.633,A -85,B 0,C 180,E1 16367.615,E2 16367.615} C_VEL
LIN {X 0,Y 337.994,Z 692.632,A -85,B 0,C 180,E1 16363.324,E2 16363.324} C_VEL
LIN {X 0,Y 338.021,Z 692.805,A -85,B 0,C 180,E1 16359.027,E2 16359.027} C_VEL
LIN {X 0,Y 339.033,Z 695.688,A -85,B 0,C 180,E1 16358.186,E2 16358.186} C_VEL
LIN {X 0,Y 341.682,Z 698.402,A -85,B 0,C 180,E1 16356.731,E2 16356.731} C_VEL
LIN {X 0,Y 342.211,Z 699.27,A -85,B 0,C 180,E1 16356.404,E2 16356.404} C_VEL
LIN {X 0,Y 344.04,Z 702.739,A -85,B 0,C 180,E1 16355.26,E2 16355.26} C_VEL
LIN {X 0,Y 345.844,Z 704.542,A -85,B 0,C 180,E1 16354.422,E2 16354.422} C_VEL
LIN {X 0,Y 348.097,Z 708.505,A -85,B 0,C 180,E1 16353.194,E2 16353.194} C_VEL
LIN {X 0,Y 349.461,Z 710.108,A -85,B 0,C 180,E1 16352.571,E2 16352.571} C_VEL
LIN {X 0,Y 351.9,Z 714.265,A -85,B 0,C 180,E1 16351.302,E2 16351.302} C_VEL
LIN {X 0,Y 356.314,Z 721.706,A -85,B 0,C 180,E1 16349.166,E2 16349.166} C_VEL
LIN {X 0,Y 361.132,Z 730.047,A -85,B 0,C 180,E1 16346.946,E2 16346.946} C_VEL
LIN {X 0,Y 368.02,Z 743.363,A -85,B 0,C 180,E1 16343.874,E2 16343.874} C_VEL
LIN {X 0,Y 374.401,Z 756.924,A -85,B 0,C 180,E1 16341.128,E2 16341.128} C_VEL
LIN {X 0,Y 381.321,Z 773.442,A -85,B 0,C 180,E1 16338.24,E2 16338.24} C_VEL
LIN {X 0,Y 383.415,Z 778.995,A -85,B 0,C 180,E1 16337.375,E2 16337.375} C_VEL
LIN {X 0,Y 386.736,Z 810.877,A -85,B 0,C 180,E1 16335.959,E2 16335.959} C_VEL
LIN {X 0,Y 376.841,Z 1041.524,A -85,B 0,C 180,E1 16331.409,E2 16331.409} C_VEL
LIN {X 0,Y 375.246,Z 1062.224,A -85,B 0,C 180,E1 16330.747,E2 16330.747} C_VEL
LIN {X 0,Y 372.917,Z 1082.922,A -85,B 0,C 180,E1 16329.801,E2 16329.801} C_VEL
LIN {X 0,Y 370.055,Z 1102.443,A -85,B 0,C 180,E1 16328.618,E2 16328.618} C_VEL
LIN {X 0,Y 366.835,Z 1120.584,A -85,B 0,C 180,E1 16327.234,E2 16327.234} C_VEL
LIN {X 0,Y 363.079,Z 1138.733,A -85,B 0,C 180,E1 16325.524,E2 16325.524} C_VEL
LIN {X 0,Y 358.98,Z 1156.408,A -85,B 0,C 180,E1 16323.468,E2 16323.468} C_VEL
LIN {X 0,Y 354.929,Z 1172.272,A -85,B 0,C 180,E1 16321.22,E2 16321.22} C_VEL
LIN {X 0,Y 351.085,Z 1186.605,A -85,B 0,C 180,E1 16318.769,E2 16318.769} C_VEL
LIN {X 0,Y 347.521,Z 1199.53,A -85,B 0,C 180,E1 16316.116,E2 16316.116} C_VEL
LIN {X 0,Y 344.188,Z 1211.7,A -85,B 0,C 180,E1 16313.089,E2 16313.089} C_VEL
LIN {X 0,Y 341.515,Z 1221.907,A -85,B 0,C 180,E1 16309.982,E2 16309.982} C_VEL
LIN {X 0,Y 339.461,Z 1230.438,A -85,B 0,C 180,E1 16306.776,E2 16306.776} C_VEL
LIN {X 0,Y 337.952,Z 1237.626,A -85,B 0,C 180,E1 16303.342,E2 16303.342} C_VEL
LIN {X 0,Y 336.994,Z 1243.207,A -85,B 0,C 180,E1 16299.736,E2 16299.736} C_VEL
LIN {X 0,Y 336.515,Z 1246.8,A -85,B 0,C 180,E1 16296.311,E2 16296.311} C_VEL
LIN {X 0,Y 336.352,Z 1248.564,A -85,B 0,C 180,E1 16293.669,E2 16293.669} C_VEL
LIN {X 0,Y 335.313,Z 1249.146,A -85,B 0,C 180,E1 16292.36,E2 16292.36} C_VEL
LIN {X 0,Y 330.684,Z 1249.918,A -85,B 0,C 180,E1 16289.883,E2 16289.883} C_VEL
LIN {X 0,Y 328.473,Z 1249.885,A -85,B 0,C 180,E1 16288.171,E2 16288.171} C_VEL
LIN {X 0,Y 328.334,Z 1249.74,A -85,B 0,C 180,E1 16287.685,E2 16287.685} C_VEL
LIN {X 0,Y 328.492,Z 1248.046,A -85,B 0,C 180,E1 16284.234,E2 16284.234} C_VEL
LIN {X 0,Y 328.92,Z 1244.751,A -85,B 0,C 180,E1 16280.728,E2 16280.728} C_VEL
LIN {X 0,Y 329.78,Z 1239.843,A -85,B 0,C 180,E1 16277.212,E2 16277.212} C_VEL
LIN {X 0,Y 331.219,Z 1233.198,A -85,B 0,C 180,E1 16273.695,E2 16273.695} C_VEL
LIN {X 0,Y 333.253,Z 1225.125,A -85,B 0,C 180,E1 16270.364,E2 16270.364} C_VEL
LIN {X 0,Y 335.857,Z 1215.688,A -85,B 0,C 180,E1 16267.23,E2 16267.23} C_VEL
LIN {X 0,Y 339.151,Z 1204.179,A -85,B 0,C 180,E1 16264.13,E2 16264.13} C_VEL
LIN {X 0,Y 342.687,Z 1191.943,A -85,B 0,C 180,E1 16261.412,E2 16261.412} C_VEL
LIN {X 0,Y 346.686,Z 1177.932,A -85,B 0,C 180,E1 16258.822,E2 16258.822} C_VEL
LIN {X 0,Y 351.061,Z 1161.793,A -85,B 0,C 180,E1 16256.36,E2 16256.36} C_VEL
LIN {X 0,Y 355.256,Z 1145.08,A -85,B 0,C 180,E1 16254.267,E2 16254.267} C_VEL
LIN {X 0,Y 359.091,Z 1128.159,A -85,B 0,C 180,E1 16252.52,E2 16252.52} C_VEL
LIN {X 0,Y 362.757,Z 1109.642,A -85,B 0,C 180,E1 16250.963,E2 16250.963} C_VEL
LIN {X 0,Y 366.017,Z 1089.855,A -85,B 0,C 180,E1 16249.652,E2 16249.652} C_VEL
LIN {X 0,Y 368.551,Z 1069.972,A -85,B 0,C 180,E1 16248.641,E2 16248.641} C_VEL
LIN {X 0,Y 370.42,Z 1049.618,A -85,B 0,C 180,E1 16247.887,E2 16247.887} C_VEL
LIN {X 0,Y 371.752,Z 1025.548,A -85,B 0,C 180,E1 16247.31,E2 16247.31} C_VEL
LIN {X 0,Y 380.667,Z 823.768,A -85,B 0,C 180,E1 16243.315,E2 16243.315} C_VEL
LIN {X 0,Y 375.438,Z 795.142,A -85,B 0,C 180,E1 16241.642,E2 16241.642} C_VEL
LIN {X 0,Y 369.857,Z 802.412,A -85,B 0,C 180,E1 16240.86,E2 16240.86} C_VEL
LIN {X 0,Y 366.368,Z 805.217,A -85,B 0,C 180,E1 16240.301,E2 16240.301} C_VEL
LIN {X 0,Y 364.435,Z 805.413,A -85,B 0,C 180,E1 16239.942,E2 16239.942} C_VEL
LIN {X 0,Y 358.507,Z 847.215,A -85,B 0,C 180,E1 16235.36,E2 16235.36} C_VEL
LIN {X 0,Y 355.399,Z 872.41,A -85,B 0,C 180,E1 16232.666,E2 16232.666} C_VEL
LIN {X 0,Y 356.244,Z 882.503,A -85,B 0,C 180,E1 16232.221,E2 16232.221} C_VEL
LIN {X 0,Y 346.543,Z 1038.333,A -85,B 0,C 180,E1 16227.621,E2 16227.621} C_VEL
LIN {X 0,Y 345.551,Z 1057.208,A -85,B 0,C 180,E1 16226.817,E2 16226.817} C_VEL
LIN {X 0,Y 344.183,Z 1074.575,A -85,B 0,C 180,E1 16225.768,E2 16225.768} C_VEL
LIN {X 0,Y 342.442,Z 1091.592,A -85,B 0,C 180,E1 16224.403,E2 16224.403} C_VEL
LIN {X 0,Y 340.457,Z 1108.022,A -85,B 0,C 180,E1 16222.727,E2 16222.727} C_VEL
LIN {X 0,Y 338.466,Z 1122.645,A -85,B 0,C 180,E1 16220.853,E2 16220.853} C_VEL
LIN {X 0,Y 336.42,Z 1136.731,A -85,B 0,C 180,E1 16218.633,E2 16218.633} C_VEL
LIN {X 0,Y 334.649,Z 1148.696,A -85,B 0,C 180,E1 16216.311,E2 16216.311} C_VEL
LIN {X 0,Y 333.057,Z 1159.488,A -85,B 0,C 180,E1 16213.72,E2 16213.72} C_VEL
LIN {X 0,Y 331.82,Z 1168.772,A -85,B 0,C 180,E1 16210.944,E2 16210.944} C_VEL
LIN {X 0,Y 331.006,Z 1176.015,A -85,B 0,C 180,E1 16208.162,E2 16208.162} C_VEL
LIN {X 0,Y 330.487,Z 1182.111,A -85,B 0,C 180,E1 16205.034,E2 16205.034} C_VEL
LIN {X 0,Y 330.334,Z 1186.09,A -85,B 0,C 180,E1 16202.082,E2 16202.082} C_VEL
LIN {X 0,Y 330.457,Z 1188.433,A -85,B 0,C 180,E1 16198.96,E2 16198.96} C_VEL
LIN {X 0,Y 330.861,Z 1189.05,A -85,B 0,C 180,E1 16195.841,E2 16195.841} C_VEL
LIN {X 0,Y 331.569,Z 1187.954,A -85,B 0,C 180,E1 16192.898,E2 16192.898} C_VEL
LIN {X 0,Y 332.817,Z 1184.851,A -85,B 0,C 180,E1 16189.616,E2 16189.616} C_VEL
LIN {X 0,Y 334.422,Z 1180.26,A -85,B 0,C 180,E1 16186.691,E2 16186.691} C_VEL
LIN {X 0,Y 336.739,Z 1173.413,A -85,B 0,C 180,E1 16183.616,E2 16183.616} C_VEL
LIN {X 0,Y 339.352,Z 1165.254,A -85,B 0,C 180,E1 16180.911,E2 16180.911} C_VEL
LIN {X 0,Y 342.305,Z 1155.719,A -85,B 0,C 180,E1 16178.406,E2 16178.406} C_VEL
LIN {X 0,Y 345.705,Z 1143.748,A -85,B 0,C 180,E1 16175.933,E2 16175.933} C_VEL
LIN {X 0,Y 349.036,Z 1130.926,A -85,B 0,C 180,E1 16173.823,E2 16173.823} C_VEL
LIN {X 0,Y 352.366,Z 1116.777,A -85,B 0,C 180,E1 16171.944,E2 16171.944} C_VEL
LIN {X 0,Y 355.672,Z 1100.848,A -85,B 0,C 180,E1 16170.253,E2 16170.253} C_VEL
LIN {X 0,Y 358.745,Z 1083.882,A -85,B 0,C 180,E1 16168.831,E2 16168.831} C_VEL
LIN {X 0,Y 363.464,Z 1061.627,A -85,B 0,C 180,E1 16167.279,E2 16167.279} C_VEL
LIN {X 0,Y 371.542,Z 1034.42,A -85,B 0,C 180,E1 16165.589,E2 16165.589} C_VEL
LIN {X 0,Y 384.529,Z 994.203,A -85,B 0,C 180,E1 16163.548,E2 16163.548} C_VEL
LIN {X 0,Y 394.747,Z 958.503,A -85,B 0,C 180,E1 16162.035,E2 16162.035} C_VEL
LIN {X 0,Y 398.041,Z 947.354,A -85,B 0,C 180,E1 16161.604,E2 16161.604} C_VEL
LIN {X 0,Y 405.083,Z 937.778,A -85,B 0,C 180,E1 16161.176,E2 16161.176} C_VEL
LIN {X 0,Y 405.524,Z 942.868,A -85,B 0,C 180,E1 16159.848,E2 16159.848} C_VEL
LIN {X 0,Y 397.564,Z 957.772,A -85,B 0,C 180,E1 16159.332,E2 16159.332} C_VEL
LIN {X 0,Y 389.182,Z 994.319,A -85,B 0,C 180,E1 16158.725,E2 16158.725} C_VEL
LIN {X 0,Y 382.79,Z 1019.347,A -85,B 0,C 180,E1 16158.279,E2 16158.279} C_VEL
LIN {X 0,Y 378.714,Z 1035.639,A -85,B 0,C 180,E1 16157.723,E2 16157.723} C_VEL
LIN {X 0,Y 371.355,Z 1066.649,A -85,B 0,C 180,E1 16156.186,E2 16156.186} C_VEL
LIN {X 0,Y 364.67,Z 1094.336,A -85,B 0,C 180,E1 16154.471,E2 16154.471} C_VEL
LIN {X 0,Y 358.687,Z 1119.712,A -85,B 0,C 180,E1 16152.531,E2 16152.531} C_VEL
LIN {X 0,Y 355.703,Z 1133.658,A -85,B 0,C 180,E1 16151.344,E2 16151.344} C_VEL
LIN {X 0,Y 353.312,Z 1152.657,A -85,B 0,C 180,E1 16149.972,E2 16149.972} C_VEL
LIN {X 0,Y 350.34,Z 1171.838,A -85,B 0,C 180,E1 16148.266,E2 16148.266} C_VEL
LIN {X 0,Y 346.922,Z 1190.724,A -85,B 0,C 180,E1 16146.216,E2 16146.216} C_VEL
LIN {X 0,Y 343.553,Z 1207.891,A -85,B 0,C 180,E1 16143.958,E2 16143.958} C_VEL
LIN {X 0,Y 340.294,Z 1223.391,A -85,B 0,C 180,E1 16141.535,E2 16141.535} C_VEL
LIN {X 0,Y 337.119,Z 1238.514,A -85,B 0,C 180,E1 16138.717,E2 16138.717} C_VEL
LIN {X 0,Y 334.372,Z 1252.063,A -85,B 0,C 180,E1 16135.696,E2 16135.696} C_VEL
LIN {X 0,Y 332.215,Z 1263.492,A -85,B 0,C 180,E1 16132.659,E2 16132.659} C_VEL
LIN {X 0,Y 330.526,Z 1273.592,A -85,B 0,C 180,E1 16129.437,E2 16129.437} C_VEL
LIN {X 0,Y 329.339,Z 1282.211,A -85,B 0,C 180,E1 16126.039,E2 16126.039} C_VEL
LIN {X 0,Y 328.696,Z 1289.024,A -85,B 0,C 180,E1 16122.652,E2 16122.652} C_VEL
LIN {X 0,Y 328.382,Z 1294.392,A -85,B 0,C 180,E1 16119.111,E2 16119.111} C_VEL
LIN {X 0,Y 328.34,Z 1297.88,A -85,B 0,C 180,E1 16115.768,E2 16115.768} C_VEL
LIN {X 0,Y 328.374,Z 1299.675,A -85,B 0,C 180,E1 16112.619,E2 16112.619} C_VEL
LIN {X 0,Y 328.385,Z 1300.113,A -85,B 0,C 180,E1 16109.303,E2 16109.303} C_VEL
LIN {X 0,Y 328.353,Z 1299.165,A -85,B 0,C 180,E1 16106.16,E2 16106.16} C_VEL
LIN {X 0,Y 328.318,Z 1296.576,A -85,B 0,C 180,E1 16102.828,E2 16102.828} C_VEL
LIN {X 0,Y 328.44,Z 1292.196,A -85,B 0,C 180,E1 16099.299,E2 16099.299} C_VEL
LIN {X 0,Y 328.827,Z 1286.379,A -85,B 0,C 180,E1 16095.922,E2 16095.922} C_VEL
LIN {X 0,Y 329.659,Z 1278.816,A -85,B 0,C 180,E1 16092.527,E2 16092.527} C_VEL
LIN {X 0,Y 331.027,Z 1269.295,A -85,B 0,C 180,E1 16089.121,E2 16089.121} C_VEL
LIN {X 0,Y 332.897,Z 1258.311,A -85,B 0,C 180,E1 16085.892,E2 16085.892} C_VEL
LIN {X 0,Y 335.28,Z 1245.928,A -85,B 0,C 180,E1 16082.854,E2 16082.854} C_VEL
LIN {X 0,Y 338.176,Z 1231.685,A -85,B 0,C 180,E1 16079.925,E2 16079.925} C_VEL
LIN {X 0,Y 341.3,Z 1216.393,A -85,B 0,C 180,E1 16077.283,E2 16077.283} C_VEL
LIN {X 0,Y 344.583,Z 1200.057,A -85,B 0,C 180,E1 16074.911,E2 16074.911} C_VEL
LIN {X 0,Y 351,Z 1170.003,A -85,B 0,C 180,E1 16071.195,E2 16071.195} C_VEL
LIN {X 0,Y 355.165,Z 1150.781,A -85,B 0,C 180,E1 16069.224,E2 16069.224} C_VEL
LIN {X 0,Y 359.796,Z 1128.281,A -85,B 0,C 180,E1 16067.308,E2 16067.308} C_VEL
LIN {X 0,Y 363.84,Z 1106.859,A -85,B 0,C 180,E1 16065.827,E2 16065.827} C_VEL
LIN {X 0,Y 367.722,Z 1083.767,A -85,B 0,C 180,E1 16064.571,E2 16064.571} C_VEL
LIN {X 0,Y 371.209,Z 1059.532,A -85,B 0,C 180,E1 16063.569,E2 16063.569} C_VEL
LIN {X 0,Y 373.449,Z 1036.469,A -85,B 0,C 180,E1 16062.863,E2 16062.863} C_VEL
LIN {X 0,Y 375.562,Z 1016.178,A -85,B 0,C 180,E1 16062.43,E2 16062.43} C_VEL
LIN {X 0,Y 377.433,Z 1003.457,A -85,B 0,C 180,E1 16062.234,E2 16062.234} C_VEL
LIN {X 0,Y 391.18,Z 972.079,A -85,B 0,C 180,E1 16060.726,E2 16060.726} C_VEL
LIN {X 0,Y 401.869,Z 951.601,A -85,B 0,C 180,E1 16059.978,E2 16059.978} C_VEL
LIN {X 0,Y 405.9,Z 943.437,A -85,B 0,C 180,E1 16059.667,E2 16059.667} C_VEL
LIN {X 0,Y 398.655,Z 926.977,A -85,B 0,C 180,E1 16057.189,E2 16057.189} C_VEL
LIN {X 0,Y 393.68,Z 909.485,A -85,B 0,C 180,E1 16054.762,E2 16054.762} C_VEL
LIN {X 0,Y 390.804,Z 890.38,A -85,B 0,C 180,E1 16052.324,E2 16052.324} C_VEL
LIN {X 0,Y 390.107,Z 869.539,A -85,B 0,C 180,E1 16049.91,E2 16049.91} C_VEL
LIN {X 0,Y 391.497,Z 848.396,A -85,B 0,C 180,E1 16047.698,E2 16047.698} C_VEL
LIN {X 0,Y 395.203,Z 824.179,A -85,B 0,C 180,E1 16045.42,E2 16045.42} C_VEL
LIN {X 0,Y 397.112,Z 813.951,A -85,B 0,C 180,E1 16044.507,E2 16044.507} C_VEL
LIN {X 0,Y 388.321,Z 796.519,A -85,B 0,C 180,E1 16040.655,E2 16040.655} C_VEL
LIN {X 0,Y 380.066,Z 780.952,A -85,B 0,C 180,E1 16036.821,E2 16036.821} C_VEL
LIN {X 0,Y 373.314,Z 768.533,A -85,B 0,C 180,E1 16033.474,E2 16033.474} C_VEL
LIN {X 0,Y 366.026,Z 755.353,A -85,B 0,C 180,E1 16029.592,E2 16029.592} C_VEL
LIN {X 0,Y 359.747,Z 744.558,A -85,B 0,C 180,E1 16026.062,E2 16026.062} C_VEL
LIN {X 0,Y 354.601,Z 735.471,A -85,B 0,C 180,E1 16022.909,E2 16022.909} C_VEL
LIN {X 0,Y 350.965,Z 729.474,A -85,B 0,C 180,E1 16020.628,E2 16020.628} C_VEL
LIN {X 0,Y 348.294,Z 724.854,A -85,B 0,C 180,E1 16018.848,E2 16018.848} C_VEL
LIN {X 0,Y 345.391,Z 719.903,A -85,B 0,C 180,E1 16016.847,E2 16016.847} C_VEL
LIN {X 0,Y 343.063,Z 715.801,A -85,B 0,C 180,E1 16015.151,E2 16015.151} C_VEL
LIN {X 0,Y 340.009,Z 710.765,A -85,B 0,C 180,E1 16012.905,E2 16012.905} C_VEL
LIN {X 0,Y 338.8,Z 709,A -85,B 0,C 180,E1 16012.027,E2 16012.027} C_VEL
LIN {X 0,Y 336.73,Z 705.207,A -85,B 0,C 180,E1 16010.331,E2 16010.331} C_VEL
LIN {X 0,Y 335.906,Z 703.999,A -85,B 0,C 180,E1 16009.712,E2 16009.712} C_VEL
LIN {X 0,Y 333.653,Z 700.368,A -85,B 0,C 180,E1 16007.891,E2 16007.891} C_VEL
LIN {X 0,Y 333.092,Z 698.954,A -85,B 0,C 180,E1 16007.304,E2 16007.304} C_VEL
LIN {X 0,Y 330.674,Z 695.854,A -85,B 0,C 180,E1 16005.465,E2 16005.465} C_VEL
LIN {X 0,Y 330.05,Z 693.617,A -85,B 0,C 180,E1 16004.538,E2 16004.538} C_VEL
LIN {X 0,Y 330.079,Z 693.803,A -85,B 0,C 180,E1 16002.367,E2 16002.367} C_VEL
LIN {X 0,Y 331.131,Z 696.742,A -85,B 0,C 180,E1 16001.332,E2 16001.332} C_VEL
LIN {X 0,Y 333.856,Z 699.467,A -85,B 0,C 180,E1 15999.671,E2 15999.671} C_VEL
LIN {X 0,Y 334.426,Z 700.037,A -85,B 0,C 180,E1 15999.341,E2 15999.341} C_VEL
LIN {X 0,Y 336.043,Z 703.418,A -85,B 0,C 180,E1 15998.165,E2 15998.165} C_VEL
LIN {X 0,Y 338.426,Z 705.789,A -85,B 0,C 180,E1 15996.862,E2 15996.862} C_VEL
LIN {X 0,Y 340.449,Z 709.693,A -85,B 0,C 180,E1 15995.537,E2 15995.537} C_VEL
LIN {X 0,Y 342.029,Z 711.444,A -85,B 0,C 180,E1 15994.735,E2 15994.735} C_VEL
LIN {X 0,Y 344.659,Z 715.795,A -85,B 0,C 180,E1 15993.278,E2 15993.278} C_VEL
LIN {X 0,Y 345.916,Z 717.794,A -85,B 0,C 180,E1 15992.639,E2 15992.639} C_VEL
LIN {X 0,Y 349.012,Z 722.863,A -85,B 0,C 180,E1 15991.042,E2 15991.042} C_VEL
LIN {X 0,Y 354.207,Z 731.78,A -85,B 0,C 180,E1 15988.481,E2 15988.481} C_VEL
LIN {X 0,Y 360.861,Z 744.341,A -85,B 0,C 180,E1 15985.376,E2 15985.376} C_VEL
LIN {X 0,Y 367.396,Z 758.028,A -85,B 0,C 180,E1 15982.438,E2 15982.438} C_VEL
LIN {X 0,Y 374.162,Z 773.842,A -85,B 0,C 180,E1 15979.506,E2 15979.506} C_VEL
LIN {X 0,Y 377.255,Z 781.252,A -85,B 0,C 180,E1 15978.324,E2 15978.324} C_VEL
LIN {X 0,Y 378.263,Z 783.551,A -85,B 0,C 180,E1 15978.086,E2 15978.086} C_VEL
LIN {X 0,Y 381.186,Z 812.288,A -85,B 0,C 180,E1 15976.803,E2 15976.803} C_VEL
LIN {X 0,Y 370.886,Z 1042.143,A -85,B 0,C 180,E1 15972.223,E2 15972.223} C_VEL
LIN {X 0,Y 369.236,Z 1062.784,A -85,B 0,C 180,E1 15971.555,E2 15971.555} C_VEL
LIN {X 0,Y 366.816,Z 1083.501,A -85,B 0,C 180,E1 15970.599,E2 15970.599} C_VEL
LIN {X 0,Y 363.842,Z 1103.031,A -85,B 0,C 180,E1 15969.404,E2 15969.404} C_VEL
LIN {X 0,Y 360.492,Z 1121.18,A -85,B 0,C 180,E1 15968.004,E2 15968.004} C_VEL
LIN {X 0,Y 356.58,Z 1139.334,A -85,B 0,C 180,E1 15966.273,E2 15966.273} C_VEL
LIN {X 0,Y 352.3,Z 1157.014,A -85,B 0,C 180,E1 15964.189,E2 15964.189} C_VEL
LIN {X 0,Y 348.065,Z 1172.881,A -85,B 0,C 180,E1 15961.907,E2 15961.907} C_VEL
LIN {X 0,Y 344.032,Z 1187.217,A -85,B 0,C 180,E1 15959.416,E2 15959.416} C_VEL
LIN {X 0,Y 340.279,Z 1200.148,A -85,B 0,C 180,E1 15956.714,E2 15956.714} C_VEL
LIN {X 0,Y 336.762,Z 1212.316,A -85,B 0,C 180,E1 15953.628,E2 15953.628} C_VEL
LIN {X 0,Y 333.87,Z 1222.721,A -85,B 0,C 180,E1 15950.386,E2 15950.386} C_VEL
LIN {X 0,Y 331.634,Z 1231.441,A -85,B 0,C 180,E1 15947.004,E2 15947.004} C_VEL
LIN {X 0,Y 330.046,Z 1238.553,A -85,B 0,C 180,E1 15943.478,E2 15943.478} C_VEL
LIN {X 0,Y 329.045,Z 1244.053,A -85,B 0,C 180,E1 15939.797,E2 15939.797} C_VEL
LIN {X 0,Y 328.545,Z 1247.563,A -85,B 0,C 180,E1 15936.289,E2 15936.289} C_VEL
LIN {X 0,Y 328.344,Z 1249.528,A -85,B 0,C 180,E1 15932.787,E2 15932.787} C_VEL
LIN {X 0,Y 328.304,Z 1250.006,A -85,B 0,C 180,E1 15929.301,E2 15929.301} C_VEL
LIN {X 0,Y 328.334,Z 1249.74,A -85,B 0,C 180,E1 15927.685,E2 15927.685} C_VEL
LIN {X 0,Y 327.37,Z 1249.339,A -85,B 0,C 180,E1 15926.341,E2 15926.341} C_VEL
LIN {X 0,Y 321.317,Z 1247.525,A -85,B 0,C 180,E1 15922.641,E2 15922.641} C_VEL
LIN {X 0,Y 320.827,Z 1246.521,A -85,B 0,C 180,E1 15921.563,E2 15921.563} C_VEL
LIN {X 0,Y 321.59,Z 1242.155,A -85,B 0,C 180,E1 15917.976,E2 15917.976} C_VEL
LIN {X 0,Y 322.949,Z 1235.951,A -85,B 0,C 180,E1 15914.338,E2 15914.338} C_VEL
LIN {X 0,Y 324.957,Z 1228.179,A -85,B 0,C 180,E1 15910.841,E2 15910.841} C_VEL
LIN {X 0,Y 327.563,Z 1219.057,A -85,B 0,C 180,E1 15907.569,E2 15907.569} C_VEL
LIN {X 0,Y 330.84,Z 1208.167,A -85,B 0,C 180,E1 15904.394,E2 15904.394} C_VEL
LIN {X 0,Y 334.637,Z 1195.817,A -85,B 0,C 180,E1 15901.44,E2 15901.44} C_VEL
LIN {X 0,Y 338.823,Z 1181.973,A -85,B 0,C 180,E1 15898.709,E2 15898.709} C_VEL
LIN {X 0,Y 343.289,Z 1166.511,A -85,B 0,C 180,E1 15896.199,E2 15896.199} C_VEL
LIN {X 0,Y 347.735,Z 1149.866,A -85,B 0,C 180,E1 15893.984,E2 15893.984} C_VEL
LIN {X 0,Y 351.824,Z 1132.884,A -85,B 0,C 180,E1 15892.13,E2 15892.13} C_VEL
LIN {X 0,Y 355.589,Z 1115.127,A -85,B 0,C 180,E1 15890.544,E2 15890.544} C_VEL
LIN {X 0,Y 359.143,Z 1095.4,A -85,B 0,C 180,E1 15889.137,E2 15889.137} C_VEL
LIN {X 0,Y 362.016,Z 1075.322,A -85,B 0,C 180,E1 15888.03,E2 15888.03} C_VEL
LIN {X 0,Y 364.126,Z 1055.509,A -85,B 0,C 180,E1 15887.219,E2 15887.219} C_VEL
LIN {X 0,Y 365.54,Z 1034.501,A -85,B 0,C 180,E1 15886.634,E2 15886.634} C_VEL
LIN {X 0,Y 375.165,Z 825.501,A -85,B 0,C 180,E1 15882.453,E2 15882.453} C_VEL
LIN {X 0,Y 372.188,Z 808.987,A -85,B 0,C 180,E1 15881.469,E2 15881.469} C_VEL
LIN {X 0,Y 367.954,Z 812.405,A -85,B 0,C 180,E1 15880.808,E2 15880.808} C_VEL
LIN {X 0,Y 366.243,Z 813.421,A -85,B 0,C 180,E1 15880.523,E2 15880.523} C_VEL
LIN {X 0,Y 361.349,Z 820.374,A -85,B 0,C 180,E1 15879.808,E2 15879.808} C_VEL
LIN {X 0,Y 357.803,Z 823.661,A -85,B 0,C 180,E1 15879.216,E2 15879.216} C_VEL
LIN {X 0,Y 355.561,Z 824.261,A -85,B 0,C 180,E1 15878.784,E2 15878.784} C_VEL
LIN {X 0,Y 349.928,Z 863.221,A -85,B 0,C 180,E1 15874.455,E2 15874.455} C_VEL
LIN {X 0,Y 348.716,Z 873.636,A -85,B 0,C 180,E1 15873.361,E2 15873.361} C_VEL
LIN {X 0,Y 349.501,Z 883.726,A -85,B 0,C 180,E1 15872.908,E2 15872.908} C_VEL
LIN {X 0,Y 339.293,Z 1038.893,A -85,B 0,C 180,E1 15868.179,E2 15868.179} C_VEL
LIN {X 0,Y 338.271,Z 1057.625,A -85,B 0,C 180,E1 15867.368,E2 15867.368} C_VEL
LIN {X 0,Y 336.882,Z 1074.869,A -85,B 0,C 180,E1 15866.319,E2 15866.319} C_VEL
LIN {X 0,Y 335.129,Z 1091.542,A -85,B 0,C 180,E1 15864.972,E2 15864.972} C_VEL
LIN {X 0,Y 333.07,Z 1108.002,A -85,B 0,C 180,E1 15863.277,E2 15863.277} C_VEL
LIN {X 0,Y 330.978,Z 1122.991,A -85,B 0,C 180,E1 15861.348,E2 15861.348} C_VEL
LIN {X 0,Y 328.832,Z 1137.203,A -85,B 0,C 180,E1 15859.079,E2 15859.079} C_VEL
LIN {X 0,Y 326.978,Z 1149.34,A -85,B 0,C 180,E1 15856.705,E2 15856.705} C_VEL
LIN {X 0,Y 325.309,Z 1160.272,A -85,B 0,C 180,E1 15854.053,E2 15854.053} C_VEL
LIN {X 0,Y 324.005,Z 1169.687,A -85,B 0,C 180,E1 15851.211,E2 15851.211} C_VEL
LIN {X 0,Y 323.153,Z 1177.09,A -85,B 0,C 180,E1 15848.362,E2 15848.362} C_VEL
LIN {X 0,Y 322.62,Z 1183.009,A -85,B 0,C 180,E1 15845.335,E2 15845.335} C_VEL
LIN {X 0,Y 322.447,Z 1187.395,A -85,B 0,C 180,E1 15842.133,E2 15842.133} C_VEL
LIN {X 0,Y 322.573,Z 1189.787,A -85,B 0,C 180,E1 15839.112,E2 15839.112} C_VEL
LIN {X 0,Y 322.992,Z 1190.599,A -85,B 0,C 180,E1 15835.918,E2 15835.918} C_VEL
LIN {X 0,Y 323.805,Z 1189.659,A -85,B 0,C 180,E1 15832.727,E2 15832.727} C_VEL
LIN {X 0,Y 325.068,Z 1186.897,A -85,B 0,C 180,E1 15829.545,E2 15829.545} C_VEL
LIN {X 0,Y 326.892,Z 1182.291,A -85,B 0,C 180,E1 15826.378,E2 15826.378} C_VEL
LIN {X 0,Y 329.37,Z 1175.624,A -85,B 0,C 180,E1 15823.239,E2 15823.239} C_VEL
LIN {X 0,Y 332.173,Z 1167.743,A -85,B 0,C 180,E1 15820.482,E2 15820.482} C_VEL
LIN {X 0,Y 335.544,Z 1157.787,A -85,B 0,C 180,E1 15817.764,E2 15817.764} C_VEL
LIN {X 0,Y 339.371,Z 1145.55,A -85,B 0,C 180,E1 15815.154,E2 15815.154} C_VEL
LIN {X 0,Y 343.236,Z 1132.031,A -85,B 0,C 180,E1 15812.878,E2 15812.878} C_VEL
LIN {X 0,Y 347.282,Z 1116.436,A -85,B 0,C 180,E1 15810.791,E2 15810.791} C_VEL
LIN {X 0,Y 351.046,Z 1100.122,A -85,B 0,C 180,E1 15809.063,E2 15809.063} C_VEL
LIN {X 0,Y 355.139,Z 1081.141,A -85,B 0,C 180,E1 15807.47,E2 15807.47} C_VEL
LIN {X 0,Y 361.246,Z 1059.745,A -85,B 0,C 180,E1 15805.911,E2 15805.911} C_VEL
LIN {X 0,Y 371.237,Z 1031.592,A -85,B 0,C 180,E1 15804.164,E2 15804.164} C_VEL
LIN {X 0,Y 383.34,Z 997.551,A -85,B 0,C 180,E1 15802.46,E2 15802.46} C_VEL
LIN {X 0,Y 393.622,Z 964.324,A -85,B 0,C 180,E1 15801.059,E2 15801.059} C_VEL
LIN {X 0,Y 397.543,Z 951.934,A -85,B 0,C 180,E1 15800.574,E2 15800.574} C_VEL
LIN {X 0,Y 386.842,Z 994.578,A -85,B 0,C 180,E1 15799.855,E2 15799.855} C_VEL
LIN {X 0,Y 379.476,Z 1020.874,A -85,B 0,C 180,E1 15799.362,E2 15799.362} C_VEL
LIN {X 0,Y 374.921,Z 1037.242,A -85,B 0,C 180,E1 15798.769,E2 15798.769} C_VEL
LIN {X 0,Y 366.401,Z 1068.985,A -85,B 0,C 180,E1 15797.114,E2 15797.114} C_VEL
LIN {X 0,Y 359.107,Z 1095.914,A -85,B 0,C 180,E1 15795.349,E2 15795.349} C_VEL
LIN {X 0,Y 352.131,Z 1122.731,A -85,B 0,C 180,E1 15793.182,E2 15793.182} C_VEL
LIN {X 0,Y 349.44,Z 1134.261,A -85,B 0,C 180,E1 15792.154,E2 15792.154} C_VEL
LIN {X 0,Y 346.706,Z 1154.119,A -85,B 0,C 180,E1 15790.672,E2 15790.672} C_VEL
LIN {X 0,Y 343.567,Z 1172.905,A -85,B 0,C 180,E1 15788.948,E2 15788.948} C_VEL
LIN {X 0,Y 339.988,Z 1191.46,A -85,B 0,C 180,E1 15786.879,E2 15786.879} C_VEL
LIN {X 0,Y 336.31,Z 1209.039,A -85,B 0,C 180,E1 15784.498,E2 15784.498} C_VEL
LIN {X 0,Y 332.65,Z 1225.361,A -85,B 0,C 180,E1 15781.838,E2 15781.838} C_VEL
LIN {X 0,Y 329.436,Z 1239.622,A -85,B 0,C 180,E1 15779.053,E2 15779.053} C_VEL
LIN {X 0,Y 326.716,Z 1252.156,A -85,B 0,C 180,E1 15776.148,E2 15776.148} C_VEL
LIN {X 0,Y 324.275,Z 1264.269,A -85,B 0,C 180,E1 15772.792,E2 15772.792} C_VEL
LIN {X 0,Y 322.49,Z 1274.412,A -85,B 0,C 180,E1 15769.375,E2 15769.375} C_VEL
LIN {X 0,Y 321.294,Z 1282.804,A -85,B 0,C 180,E1 15765.894,E2 15765.894} C_VEL
LIN {X 0,Y 320.638,Z 1289.674,A -85,B 0,C 180,E1 15762.243,E2 15762.243} C_VEL
LIN {X 0,Y 320.379,Z 1294.43,A -85,B 0,C 180,E1 15758.797,E2 15758.797} C_VEL
LIN {X 0,Y 320.363,Z 1297.631,A -85,B 0,C 180,E1 15755.373,E2 15755.373} C_VEL
LIN {X 0,Y 320.403,Z 1299.332,A -85,B 0,C 180,E1 15751.968,E2 15751.968} C_VEL
LIN {X 0,Y 320.406,Z 1299.432,A -85,B 0,C 180,E1 15748.749,E2 15748.749} C_VEL
LIN {X 0,Y 320.362,Z 1298.109,A -85,B 0,C 180,E1 15745.346,E2 15745.346} C_VEL
LIN {X 0,Y 320.338,Z 1295.28,A -85,B 0,C 180,E1 15741.927,E2 15741.927} C_VEL
LIN {X 0,Y 320.502,Z 1290.773,A -85,B 0,C 180,E1 15738.484,E2 15738.484} C_VEL
LIN {X 0,Y 321.019,Z 1284.433,A -85,B 0,C 180,E1 15734.913,E2 15734.913} C_VEL
LIN {X 0,Y 322.046,Z 1276.301,A -85,B 0,C 180,E1 15731.351,E2 15731.351} C_VEL
LIN {X 0,Y 323.637,Z 1266.668,A -85,B 0,C 180,E1 15727.946,E2 15727.946} C_VEL
LIN {X 0,Y 325.861,Z 1255.005,A -85,B 0,C 180,E1 15724.561,E2 15724.561} C_VEL
LIN {X 0,Y 328.544,Z 1242.117,A -85,B 0,C 180,E1 15721.459,E2 15721.459} C_VEL
LIN {X 0,Y 331.728,Z 1227.56,A -85,B 0,C 180,E1 15718.537,E2 15718.537} C_VEL
LIN {X 0,Y 335.058,Z 1212.361,A -85,B 0,C 180,E1 15715.978,E2 15715.978} C_VEL
LIN {X 0,Y 338.594,Z 1195.504,A -85,B 0,C 180,E1 15713.592,E2 15713.592} C_VEL
LIN {X 0,Y 342.097,Z 1177.699,A -85,B 0,C 180,E1 15711.499,E2 15711.499} C_VEL
LIN {X 0,Y 347.995,Z 1150.597,A -85,B 0,C 180,E1 15708.638,E2 15708.638} C_VEL
LIN {X 0,Y 352.762,Z 1128.335,A -85,B 0,C 180,E1 15706.693,E2 15706.693} C_VEL
LIN {X 0,Y 357.109,Z 1106.18,A -85,B 0,C 180,E1 15705.126,E2 15705.126} C_VEL
LIN {X 0,Y 361.219,Z 1082.648,A -85,B 0,C 180,E1 15703.827,E2 15703.827} C_VEL
LIN {X 0,Y 364.83,Z 1058.299,A -85,B 0,C 180,E1 15702.805,E2 15702.805} C_VEL
LIN {X 0,Y 367.162,Z 1035.089,A -85,B 0,C 180,E1 15702.081,E2 15702.081} C_VEL
LIN {X 0,Y 369.54,Z 1013.984,A -85,B 0,C 180,E1 15701.639,E2 15701.639} C_VEL
LIN {X 0,Y 371.457,Z 1002.038,A -85,B 0,C 180,E1 15701.442,E2 15701.442} C_VEL
LIN {X 0,Y 385.338,Z 970.885,A -85,B 0,C 180,E1 15699.938,E2 15699.938} C_VEL
LIN {X 0,Y 396.072,Z 950.421,A -85,B 0,C 180,E1 15699.196,E2 15699.196} C_VEL
LIN {X 0,Y 398.503,Z 945.793,A -85,B 0,C 180,E1 15699.033,E2 15699.033} C_VEL
LIN {X 0,Y 391.741,Z 929.51,A -85,B 0,C 180,E1 15696.582,E2 15696.582} C_VEL
LIN {X 0,Y 387.124,Z 912.263,A -85,B 0,C 180,E1 15694.177,E2 15694.177} C_VEL
LIN {X 0,Y 384.42,Z 892.923,A -85,B 0,C 180,E1 15691.694,E2 15691.694} C_VEL
LIN {X 0,Y 383.931,Z 872.141,A -85,B 0,C 180,E1 15689.26,E2 15689.26} C_VEL
LIN {X 0,Y 385.532,Z 850.731,A -85,B 0,C 180,E1 15686.991,E2 15686.991} C_VEL
LIN {X 0,Y 389.451,Z 826.077,A -85,B 0,C 180,E1 15684.656,E2 15684.656} C_VEL
LIN {X 0,Y 390.96,Z 818.001,A -85,B 0,C 180,E1 15683.913,E2 15683.913} C_VEL
LIN {X 0,Y 382.249,Z 800.771,A -85,B 0,C 180,E1 15680.039,E2 15680.039} C_VEL
LIN {X 0,Y 373.752,Z 784.59,A -85,B 0,C 180,E1 15675.994,E2 15675.994} C_VEL
LIN {X 0,Y 365.992,Z 770.363,A -85,B 0,C 180,E1 15672.039,E2 15672.039} C_VEL
LIN {X 0,Y 358.401,Z 756.739,A -85,B 0,C 180,E1 15667.857,E2 15667.857} C_VEL
LIN {X 0,Y 352.228,Z 746.088,A -85,B 0,C 180,E1 15664.232,E2 15664.232} C_VEL
LIN {X 0,Y 348.833,Z 740.323,A -85,B 0,C 180,E1 15662.135,E2 15662.135} C_VEL
LIN {X 0,Y 345.948,Z 735.39,A -85,B 0,C 180,E1 15660.266,E2 15660.266} C_VEL
LIN {X 0,Y 343.351,Z 730.884,A -85,B 0,C 180,E1 15658.498,E2 15658.498} C_VEL
LIN {X 0,Y 340.434,Z 725.931,A -85,B 0,C 180,E1 15656.464,E2 15656.464} C_VEL
LIN {X 0,Y 337.574,Z 720.996,A -85,B 0,C 180,E1 15654.37,E2 15654.37} C_VEL
LIN {X 0,Y 335.125,Z 716.559,A -85,B 0,C 180,E1 15652.456,E2 15652.456} C_VEL
LIN {X 0,Y 332.248,Z 712.138,A -85,B 0,C 180,E1 15650.298,E2 15650.298} C_VEL
LIN {X 0,Y 331.36,Z 710.534,A -85,B 0,C 180,E1 15649.569,E2 15649.569} C_VEL
LIN {X 0,Y 329.064,Z 706.913,A -85,B 0,C 180,E1 15647.719,E2 15647.719} C_VEL
LIN {X 0,Y 328.283,Z 705.28,A -85,B 0,C 180,E1 15646.974,E2 15646.974} C_VEL
LIN {X 0,Y 325.914,Z 701.902,A -85,B 0,C 180,E1 15645.066,E2 15645.066} C_VEL
LIN {X 0,Y 325.205,Z 699.978,A -85,B 0,C 180,E1 15644.221,E2 15644.221} C_VEL
LIN {X 0,Y 325.047,Z 699.856,A -85,B 0,C 180,E1 15643.928,E2 15643.928} C_VEL
LIN {X 0,Y 326.816,Z 700.979,A -85,B 0,C 180,E1 15642.736,E2 15642.736} C_VEL
LIN {X 0,Y 328.257,Z 704.427,A -85,B 0,C 180,E1 15641.347,E2 15641.347} C_VEL
LIN {X 0,Y 330.888,Z 707.129,A -85,B 0,C 180,E1 15639.665,E2 15639.665} C_VEL
LIN {X 0,Y 332.795,Z 710.724,A -85,B 0,C 180,E1 15638.312,E2 15638.312} C_VEL
LIN {X 0,Y 334.864,Z 712.902,A -85,B 0,C 180,E1 15637.159,E2 15637.159} C_VEL
LIN {X 0,Y 337.196,Z 717.023,A -85,B 0,C 180,E1 15635.659,E2 15635.659} C_VEL
LIN {X 0,Y 338.405,Z 718.552,A -85,B 0,C 180,E1 15635.006,E2 15635.006} C_VEL
LIN {X 0,Y 341.872,Z 724.261,A -85,B 0,C 180,E1 15633.043,E2 15633.043} C_VEL
LIN {X 0,Y 344.867,Z 729.319,A -85,B 0,C 180,E1 15631.42,E2 15631.42} C_VEL
LIN {X 0,Y 350.214,Z 738.776,A -85,B 0,C 180,E1 15628.694,E2 15628.694} C_VEL
LIN {X 0,Y 356.11,Z 750.101,A -85,B 0,C 180,E1 15625.837,E2 15625.837} C_VEL
LIN {X 0,Y 362.578,Z 763.882,A -85,B 0,C 180,E1 15622.839,E2 15622.839} C_VEL
LIN {X 0,Y 369.287,Z 779.765,A -85,B 0,C 180,E1 15619.879,E2 15619.879} C_VEL
LIN {X 0,Y 371.796,Z 784.625,A -85,B 0,C 180,E1 15619.194,E2 15619.194} C_VEL
LIN {X 0,Y 373.212,Z 787.657,A -85,B 0,C 180,E1 15618.851,E2 15618.851} C_VEL
LIN {X 0,Y 375.722,Z 813.661,A -85,B 0,C 180,E1 15617.673,E2 15617.673} C_VEL
LIN {X 0,Y 365.002,Z 1042.864,A -85,B 0,C 180,E1 15613.06,E2 15613.06} C_VEL
LIN {X 0,Y 363.289,Z 1063.467,A -85,B 0,C 180,E1 15612.385,E2 15612.385} C_VEL
LIN {X 0,Y 360.889,Z 1083.363,A -85,B 0,C 180,E1 15611.464,E2 15611.464} C_VEL
LIN {X 0,Y 357.918,Z 1102.42,A -85,B 0,C 180,E1 15610.302,E2 15610.302} C_VEL
LIN {X 0,Y 354.321,Z 1121.3,A -85,B 0,C 180,E1 15608.845,E2 15608.845} C_VEL
LIN {X 0,Y 350.324,Z 1139.168,A -85,B 0,C 180,E1 15607.13,E2 15607.13} C_VEL
LIN {X 0,Y 346.002,Z 1156.325,A -85,B 0,C 180,E1 15605.103,E2 15605.103} C_VEL
LIN {X 0,Y 341.735,Z 1171.768,A -85,B 0,C 180,E1 15602.889,E2 15602.889} C_VEL
LIN {X 0,Y 337.548,Z 1186.038,A -85,B 0,C 180,E1 15600.431,E2 15600.431} C_VEL
LIN {X 0,Y 333.544,Z 1199.271,A -85,B 0,C 180,E1 15597.686,E2 15597.686} C_VEL
LIN {X 0,Y 329.947,Z 1211.098,A -85,B 0,C 180,E1 15594.719,E2 15594.719} C_VEL
LIN {X 0,Y 326.857,Z 1221.511,A -85,B 0,C 180,E1 15591.535,E2 15591.535} C_VEL
LIN {X 0,Y 324.245,Z 1230.862,A -85,B 0,C 180,E1 15587.96,E2 15587.96} C_VEL
LIN {X 0,Y 322.419,Z 1238.191,A -85,B 0,C 180,E1 15584.364,E2 15584.364} C_VEL
LIN {X 0,Y 321.279,Z 1243.711,A -85,B 0,C 180,E1 15580.761,E2 15580.761} C_VEL
LIN {X 0,Y 320.666,Z 1247.57,A -85,B 0,C 180,E1 15577.164,E2 15577.164} C_VEL
LIN {X 0,Y 320.397,Z 1249.881,A -85,B 0,C 180,E1 15573.578,E2 15573.578} C_VEL
LIN {X 0,Y 320.339,Z 1250.688,A -85,B 0,C 180,E1 15569.999,E2 15569.999} C_VEL
LIN {X 0,Y 320.393,Z 1249.917,A -85,B 0,C 180,E1 15566.421,E2 15566.421} C_VEL
LIN {X 0,Y 320.659,Z 1247.656,A -85,B 0,C 180,E1 15562.834,E2 15562.834} C_VEL
LIN {X 0,Y 320.827,Z 1246.521,A -85,B 0,C 180,E1 15561.563,E2 15561.563} C_VEL
LIN {X 0,Y 320.071,Z 1245.162,A -85,B 0,C 180,E1 15560.203,E2 15560.203} C_VEL
LIN {X 0,Y 314.835,Z 1241.071,A -85,B 0,C 180,E1 15556.551,E2 15556.551} C_VEL
LIN {X 0,Y 314.537,Z 1239.194,A -85,B 0,C 180,E1 15555.384,E2 15555.384} C_VEL
LIN {X 0,Y 316.519,Z 1231.709,A -85,B 0,C 180,E1 15551.585,E2 15551.585} C_VEL
LIN {X 0,Y 319.279,Z 1222.404,A -85,B 0,C 180,E1 15547.926,E2 15547.926} C_VEL
LIN {X 0,Y 322.738,Z 1211.425,A -85,B 0,C 180,E1 15544.492,E2 15544.492} C_VEL
LIN {X 0,Y 326.56,Z 1199.53,A -85,B 0,C 180,E1 15541.468,E2 15541.468} C_VEL
LIN {X 0,Y 330.787,Z 1186.221,A -85,B 0,C 180,E1 15538.674,E2 15538.674} C_VEL
LIN {X 0,Y 335.326,Z 1171.427,A -85,B 0,C 180,E1 15536.11,E2 15536.11} C_VEL
LIN {X 0,Y 340.016,Z 1155.001,A -85,B 0,C 180,E1 15533.767,E2 15533.767} C_VEL
LIN {X 0,Y 344.385,Z 1138.204,A -85,B 0,C 180,E1 15531.8,E2 15531.8} C_VEL
LIN {X 0,Y 348.463,Z 1120.581,A -85,B 0,C 180,E1 15530.111,E2 15530.111} C_VEL
LIN {X 0,Y 352.318,Z 1100.918,A -85,B 0,C 180,E1 15528.605,E2 15528.605} C_VEL
LIN {X 0,Y 355.552,Z 1080.318,A -85,B 0,C 180,E1 15527.385,E2 15527.385} C_VEL
LIN {X 0,Y 357.905,Z 1060.25,A -85,B 0,C 180,E1 15526.505,E2 15526.505} C_VEL
LIN {X 0,Y 359.48,Z 1039.984,A -85,B 0,C 180,E1 15525.884,E2 15525.884} C_VEL
LIN {X 0,Y 369.745,Z 827.172,A -85,B 0,C 180,E1 15521.562,E2 15521.562} C_VEL
LIN {X 0,Y 368.504,Z 820.495,A -85,B 0,C 180,E1 15521.146,E2 15521.146} C_VEL
LIN {X 0,Y 363.336,Z 827.274,A -85,B 0,C 180,E1 15520.397,E2 15520.397} C_VEL
LIN {X 0,Y 358.995,Z 831.019,A -85,B 0,C 180,E1 15519.68,E2 15519.68} C_VEL
LIN {X 0,Y 357.227,Z 832.188,A -85,B 0,C 180,E1 15519.369,E2 15519.369} C_VEL
LIN {X 0,Y 352.23,Z 839.589,A -85,B 0,C 180,E1 15518.594,E2 15518.594} C_VEL
LIN {X 0,Y 348.496,Z 843.278,A -85,B 0,C 180,E1 15517.93,E2 15517.93} C_VEL
LIN {X 0,Y 346.462,Z 843.924,A -85,B 0,C 180,E1 15517.512,E2 15517.512} C_VEL
LIN {X 0,Y 346.186,Z 844.06,A -85,B 0,C 180,E1 15517.433,E2 15517.433} C_VEL
LIN {X 0,Y 342.009,Z 874.688,A -85,B 0,C 180,E1 15514.075,E2 15514.075} C_VEL
LIN {X 0,Y 342.751,Z 884.689,A -85,B 0,C 180,E1 15513.61,E2 15513.61} C_VEL
LIN {X 0,Y 332.096,Z 1038.546,A -85,B 0,C 180,E1 15508.786,E2 15508.786} C_VEL
LIN {X 0,Y 331.055,Z 1057.159,A -85,B 0,C 180,E1 15507.978,E2 15507.978} C_VEL
LIN {X 0,Y 329.561,Z 1075.108,A -85,B 0,C 180,E1 15506.876,E2 15506.876} C_VEL
LIN {X 0,Y 327.718,Z 1092.212,A -85,B 0,C 180,E1 15505.48,E2 15505.48} C_VEL
LIN {X 0,Y 325.553,Z 1108.963,A -85,B 0,C 180,E1 15503.725,E2 15503.725} C_VEL
LIN {X 0,Y 323.413,Z 1123.859,A -85,B 0,C 180,E1 15501.777,E2 15501.777} C_VEL
LIN {X 0,Y 321.261,Z 1137.644,A -85,B 0,C 180,E1 15499.547,E2 15499.547} C_VEL
LIN {X 0,Y 319.318,Z 1149.933,A -85,B 0,C 180,E1 15497.118,E2 15497.118} C_VEL
LIN {X 0,Y 317.678,Z 1160.409,A -85,B 0,C 180,E1 15494.584,E2 15494.584} C_VEL
LIN {X 0,Y 316.267,Z 1170.052,A -85,B 0,C 180,E1 15491.674,E2 15491.674} C_VEL
LIN {X 0,Y 315.298,Z 1178.133,A -85,B 0,C 180,E1 15488.572,E2 15488.572} C_VEL
LIN {X 0,Y 314.736,Z 1184.166,A -85,B 0,C 180,E1 15485.469,E2 15485.469} C_VEL
LIN {X 0,Y 314.556,Z 1188.677,A -85,B 0,C 180,E1 15482.186,E2 15482.186} C_VEL
LIN {X 0,Y 314.703,Z 1191.221,A -85,B 0,C 180,E1 15479.09,E2 15479.09} C_VEL
LIN {X 0,Y 315.16,Z 1192.155,A -85,B 0,C 180,E1 15475.816,E2 15475.816} C_VEL
LIN {X 0,Y 316.049,Z 1191.383,A -85,B 0,C 180,E1 15472.548,E2 15472.548} C_VEL
LIN {X 0,Y 317.507,Z 1188.573,A -85,B 0,C 180,E1 15469.109,E2 15469.109} C_VEL
LIN {X 0,Y 319.387,Z 1184.347,A -85,B 0,C 180,E1 15466.044,E2 15466.044} C_VEL
LIN {X 0,Y 322.038,Z 1177.915,A -85,B 0,C 180,E1 15462.846,E2 15462.846} C_VEL
LIN {X 0,Y 325.033,Z 1170.295,A -85,B 0,C 180,E1 15460.035,E2 15460.035} C_VEL
LIN {X 0,Y 328.617,Z 1160.654,A -85,B 0,C 180,E1 15457.269,E2 15457.269} C_VEL
LIN {X 0,Y 332.234,Z 1150.184,A -85,B 0,C 180,E1 15454.892,E2 15454.892} C_VEL
LIN {X 0,Y 336.046,Z 1138.502,A -85,B 0,C 180,E1 15452.729,E2 15452.729} C_VEL
LIN {X 0,Y 340.273,Z 1124.33,A -85,B 0,C 180,E1 15450.613,E2 15450.613} C_VEL
LIN {X 0,Y 344.629,Z 1108.51,A -85,B 0,C 180,E1 15448.713,E2 15448.713} C_VEL
LIN {X 0,Y 349.131,Z 1091.025,A -85,B 0,C 180,E1 15447.035,E2 15447.035} C_VEL
LIN {X 0,Y 354.906,Z 1072.194,A -85,B 0,C 180,E1 15445.51,E2 15445.51} C_VEL
LIN {X 0,Y 364.985,Z 1046.379,A -85,B 0,C 180,E1 15443.721,E2 15443.721} C_VEL
LIN {X 0,Y 376.912,Z 1016.885,A -85,B 0,C 180,E1 15442.113,E2 15442.113} C_VEL
LIN {X 0,Y 385.456,Z 993.698,A -85,B 0,C 180,E1 15441.028,E2 15441.028} C_VEL
LIN {X 0,Y 377.684,Z 1019.434,A -85,B 0,C 180,E1 15440.567,E2 15440.567} C_VEL
LIN {X 0,Y 372.606,Z 1035.738,A -85,B 0,C 180,E1 15440.007,E2 15440.007} C_VEL
LIN {X 0,Y 363.846,Z 1064.737,A -85,B 0,C 180,E1 15438.491,E2 15438.491} C_VEL
LIN {X 0,Y 355.129,Z 1093.313,A -85,B 0,C 180,E1 15436.609,E2 15436.609} C_VEL
LIN {X 0,Y 347.653,Z 1119.04,A -85,B 0,C 180,E1 15434.5,E2 15434.5} C_VEL
LIN {X 0,Y 343.223,Z 1135.163,A -85,B 0,C 180,E1 15432.976,E2 15432.976} C_VEL
LIN {X 0,Y 340.163,Z 1155.524,A -85,B 0,C 180,E1 15431.404,E2 15431.404} C_VEL
LIN {X 0,Y 336.618,Z 1175.105,A -85,B 0,C 180,E1 15429.534,E2 15429.534} C_VEL
LIN {X 0,Y 332.901,Z 1192.964,A -85,B 0,C 180,E1 15427.46,E2 15427.46} C_VEL
LIN {X 0,Y 329.2,Z 1209.567,A -85,B 0,C 180,E1 15425.139,E2 15425.139} C_VEL
LIN {X 0,Y 325.347,Z 1225.747,A -85,B 0,C 180,E1 15422.431,E2 15422.431} C_VEL
LIN {X 0,Y 321.766,Z 1240.729,A -85,B 0,C 180,E1 15419.405,E2 15419.405} C_VEL
LIN {X 0,Y 318.742,Z 1253.828,A -85,B 0,C 180,E1 15416.215,E2 15416.215} C_VEL
LIN {X 0,Y 316.305,Z 1265.205,A -85,B 0,C 180,E1 15412.881,E2 15412.881} C_VEL
LIN {X 0,Y 314.453,Z 1275.217,A -85,B 0,C 180,E1 15409.311,E2 15409.311} C_VEL
LIN {X 0,Y 313.201,Z 1283.66,A -85,B 0,C 180,E1 15405.556,E2 15405.556} C_VEL
LIN {X 0,Y 312.605,Z 1289.891,A -85,B 0,C 180,E1 15402,E2 15402} C_VEL
LIN {X 0,Y 312.376,Z 1294.466,A -85,B 0,C 180,E1 15398.468,E2 15398.468} C_VEL
LIN {X 0,Y 312.38,Z 1297.261,A -85,B 0,C 180,E1 15395.143,E2 15395.143} C_VEL
LIN {X 0,Y 312.425,Z 1298.774,A -85,B 0,C 180,E1 15391.651,E2 15391.651} C_VEL
LIN {X 0,Y 312.424,Z 1298.798,A -85,B 0,C 180,E1 15388.534,E2 15388.534} C_VEL
LIN {X 0,Y 312.372,Z 1297.377,A -85,B 0,C 180,E1 15385.043,E2 15385.043} C_VEL
LIN {X 0,Y 312.352,Z 1294.458,A -85,B 0,C 180,E1 15381.533,E2 15381.533} C_VEL
LIN {X 0,Y 312.55,Z 1289.884,A -85,B 0,C 180,E1 15377.999,E2 15377.999} C_VEL
LIN {X 0,Y 313.114,Z 1283.648,A -85,B 0,C 180,E1 15374.442,E2 15374.442} C_VEL
LIN {X 0,Y 314.296,Z 1275.193,A -85,B 0,C 180,E1 15370.68,E2 15370.68} C_VEL
LIN {X 0,Y 316.096,Z 1265.168,A -85,B 0,C 180,E1 15367.105,E2 15367.105} C_VEL
LIN {X 0,Y 318.348,Z 1254.371,A -85,B 0,C 180,E1 15363.916,E2 15363.916} C_VEL
LIN {X 0,Y 321.404,Z 1240.75,A -85,B 0,C 180,E1 15360.581,E2 15360.581} C_VEL
LIN {X 0,Y 324.806,Z 1226.14,A -85,B 0,C 180,E1 15357.615,E2 15357.615} C_VEL
LIN {X 0,Y 328.462,Z 1210.514,A -85,B 0,C 180,E1 15354.969,E2 15354.969} C_VEL
LIN {X 0,Y 332.121,Z 1194.064,A -85,B 0,C 180,E1 15352.634,E2 15352.634} C_VEL
LIN {X 0,Y 335.834,Z 1176.263,A -85,B 0,C 180,E1 15350.534,E2 15350.534} C_VEL
LIN {X 0,Y 339.206,Z 1158.238,A -85,B 0,C 180,E1 15348.774,E2 15348.774} C_VEL
LIN {X 0,Y 345.334,Z 1130.175,A -85,B 0,C 180,E1 15346.214,E2 15346.214} C_VEL
LIN {X 0,Y 349.998,Z 1107.389,A -85,B 0,C 180,E1 15344.541,E2 15344.541} C_VEL
LIN {X 0,Y 354.243,Z 1084.358,A -85,B 0,C 180,E1 15343.206,E2 15343.206} C_VEL
LIN {X 0,Y 358.057,Z 1060.004,A -85,B 0,C 180,E1 15342.139,E2 15342.139} C_VEL
LIN {X 0,Y 360.69,Z 1035.954,A -85,B 0,C 180,E1 15341.348,E2 15341.348} C_VEL
LIN {X 0,Y 363.097,Z 1014.901,A -85,B 0,C 180,E1 15340.883,E2 15340.883} C_VEL
LIN {X 0,Y 365.178,Z 1001.415,A -85,B 0,C 180,E1 15340.676,E2 15340.676} C_VEL
LIN {X 0,Y 379.153,Z 970.379,A -85,B 0,C 180,E1 15339.169,E2 15339.169} C_VEL
LIN {X 0,Y 390.352,Z 949.244,A -85,B 0,C 180,E1 15338.392,E2 15338.392} C_VEL
LIN {X 0,Y 391.093,Z 947.95,A -85,B 0,C 180,E1 15338.352,E2 15338.352} C_VEL
LIN {X 0,Y 384.468,Z 930.718,A -85,B 0,C 180,E1 15335.769,E2 15335.769} C_VEL
LIN {X 0,Y 380.268,Z 913.232,A -85,B 0,C 180,E1 15333.335,E2 15333.335} C_VEL
LIN {X 0,Y 378.006,Z 894.099,A -85,B 0,C 180,E1 15330.873,E2 15330.873} C_VEL
LIN {X 0,Y 377.871,Z 872.645,A -85,B 0,C 180,E1 15328.357,E2 15328.357} C_VEL
LIN {X 0,Y 379.785,Z 851.096,A -85,B 0,C 180,E1 15326.082,E2 15326.082} C_VEL
LIN {X 0,Y 384.106,Z 826.037,A -85,B 0,C 180,E1 15323.706,E2 15323.706} C_VEL
LIN {X 0,Y 384.803,Z 822.21,A -85,B 0,C 180,E1 15323.344,E2 15323.344} C_VEL
LIN {X 0,Y 376.458,Z 805.577,A -85,B 0,C 180,E1 15319.551,E2 15319.551} C_VEL
LIN {X 0,Y 368.609,Z 790.492,A -85,B 0,C 180,E1 15315.738,E2 15315.738} C_VEL
LIN {X 0,Y 361.032,Z 776.494,A -85,B 0,C 180,E1 15311.826,E2 15311.826} C_VEL
LIN {X 0,Y 353.511,Z 762.925,A -85,B 0,C 180,E1 15307.639,E2 15307.639} C_VEL
LIN {X 0,Y 347.022,Z 751.749,A -85,B 0,C 180,E1 15303.799,E2 15303.799} C_VEL
LIN {X 0,Y 342.207,Z 743.152,A -85,B 0,C 180,E1 15300.669,E2 15300.669} C_VEL
LIN {X 0,Y 338.08,Z 736.439,A -85,B 0,C 180,E1 15297.966,E2 15297.966} C_VEL
LIN {X 0,Y 335.669,Z 732.228,A -85,B 0,C 180,E1 15296.239,E2 15296.239} C_VEL
LIN {X 0,Y 332.728,Z 727.182,A -85,B 0,C 180,E1 15294.069,E2 15294.069} C_VEL
LIN {X 0,Y 329.774,Z 722.15,A -85,B 0,C 180,E1 15291.807,E2 15291.807} C_VEL
LIN {X 0,Y 327.3,Z 717.803,A -85,B 0,C 180,E1 15289.794,E2 15289.794} C_VEL
LIN {X 0,Y 324.286,Z 712.986,A -85,B 0,C 180,E1 15287.355,E2 15287.355} C_VEL
LIN {X 0,Y 323.423,Z 711.509,A -85,B 0,C 180,E1 15286.593,E2 15286.593} C_VEL
LIN {X 0,Y 321.139,Z 707.759,A -85,B 0,C 180,E1 15284.561,E2 15284.561} C_VEL
LIN {X 0,Y 322.284,Z 707.377,A -85,B 0,C 180,E1 15283.971,E2 15283.971} C_VEL
LIN {X 0,Y 323.73,Z 708.585,A -85,B 0,C 180,E1 15282.937,E2 15282.937} C_VEL
LIN {X 0,Y 325.458,Z 712.085,A -85,B 0,C 180,E1 15281.367,E2 15281.367} C_VEL
LIN {X 0,Y 327.511,Z 714.212,A -85,B 0,C 180,E1 15280.005,E2 15280.005} C_VEL
LIN {X 0,Y 329.586,Z 718.034,A -85,B 0,C 180,E1 15278.464,E2 15278.464} C_VEL
LIN {X 0,Y 331.416,Z 720.192,A -85,B 0,C 180,E1 15277.393,E2 15277.393} C_VEL
LIN {X 0,Y 333.907,Z 724.324,A -85,B 0,C 180,E1 15275.78,E2 15275.78} C_VEL
LIN {X 0,Y 337.839,Z 730.724,A -85,B 0,C 180,E1 15273.455,E2 15273.455} C_VEL
LIN {X 0,Y 342.984,Z 739.547,A -85,B 0,C 180,E1 15270.647,E2 15270.647} C_VEL
LIN {X 0,Y 349.866,Z 752.659,A -85,B 0,C 180,E1 15267.112,E2 15267.112} C_VEL
LIN {X 0,Y 356.572,Z 766.856,A -85,B 0,C 180,E1 15263.858,E2 15263.858} C_VEL
LIN {X 0,Y 363.253,Z 782.386,A -85,B 0,C 180,E1 15260.875,E2 15260.875} C_VEL
LIN {X 0,Y 368.217,Z 791.655,A -85,B 0,C 180,E1 15259.643,E2 15259.643} C_VEL
LIN {X 0,Y 370.353,Z 814.89,A -85,B 0,C 180,E1 15258.571,E2 15258.571} C_VEL
LIN {X 0,Y 359.204,Z 1043.486,A -85,B 0,C 180,E1 15253.927,E2 15253.927} C_VEL
LIN {X 0,Y 357.42,Z 1064.153,A -85,B 0,C 180,E1 15253.243,E2 15253.243} C_VEL
LIN {X 0,Y 354.8,Z 1084.924,A -85,B 0,C 180,E1 15252.263,E2 15252.263} C_VEL
LIN {X 0,Y 351.632,Z 1104.208,A -85,B 0,C 180,E1 15251.058,E2 15251.058} C_VEL
LIN {X 0,Y 348.012,Z 1122.371,A -85,B 0,C 180,E1 15249.628,E2 15249.628} C_VEL
LIN {X 0,Y 343.777,Z 1140.536,A -85,B 0,C 180,E1 15247.855,E2 15247.855} C_VEL
LIN {X 0,Y 339.118,Z 1158.225,A -85,B 0,C 180,E1 15245.716,E2 15245.716} C_VEL
LIN {X 0,Y 334.5,Z 1174.099,A -85,B 0,C 180,E1 15243.366,E2 15243.366} C_VEL
LIN {X 0,Y 330.062,Z 1188.442,A -85,B 0,C 180,E1 15240.793,E2 15240.793} C_VEL
LIN {X 0,Y 325.923,Z 1201.373,A -85,B 0,C 180,E1 15237.992,E2 15237.992} C_VEL
LIN {X 0,Y 322.009,Z 1213.548,A -85,B 0,C 180,E1 15234.782,E2 15234.782} C_VEL
LIN {X 0,Y 318.864,Z 1223.621,A -85,B 0,C 180,E1 15231.522,E2 15231.522} C_VEL
LIN {X 0,Y 316.333,Z 1232.287,A -85,B 0,C 180,E1 15228.044,E2 15228.044} C_VEL
LIN {X 0,Y 314.464,Z 1239.473,A -85,B 0,C 180,E1 15224.359,E2 15224.359} C_VEL
LIN {X 0,Y 313.259,Z 1245.048,A -85,B 0,C 180,E1 15220.481,E2 15220.481} C_VEL
LIN {X 0,Y 312.654,Z 1248.634,A -85,B 0,C 180,E1 15216.795,E2 15216.795} C_VEL
LIN {X 0,Y 312.401,Z 1250.704,A -85,B 0,C 180,E1 15213.054,E2 15213.054} C_VEL
LIN {X 0,Y 312.351,Z 1251.245,A -85,B 0,C 180,E1 15209.449,E2 15209.449} C_VEL
LIN {X 0,Y 312.451,Z 1250.331,A -85,B 0,C 180,E1 15205.778,E2 15205.778} C_VEL
LIN {X 0,Y 312.78,Z 1247.816,A -85,B 0,C 180,E1 15202.098,E2 15202.098} C_VEL
LIN {X 0,Y 313.51,Z 1243.73,A -85,B 0,C 180,E1 15198.408,E2 15198.408} C_VEL
LIN {X 0,Y 314.537,Z 1239.194,A -85,B 0,C 180,E1 15195.384,E2 15195.384} C_VEL
LIN {X 0,Y 314.152,Z 1236.918,A -85,B 0,C 180,E1 15194.038,E2 15194.038} C_VEL
LIN {X 0,Y 310.192,Z 1230.887,A -85,B 0,C 180,E1 15190.583,E2 15190.583} C_VEL
LIN {X 0,Y 310.201,Z 1227.967,A -85,B 0,C 180,E1 15189.246,E2 15189.246} C_VEL
LIN {X 0,Y 313.416,Z 1218.078,A -85,B 0,C 180,E1 15185.698,E2 15185.698} C_VEL
LIN {X 0,Y 317.024,Z 1207.36,A -85,B 0,C 180,E1 15182.582,E2 15182.582} C_VEL
LIN {X 0,Y 321.344,Z 1194.581,A -85,B 0,C 180,E1 15179.524,E2 15179.524} C_VEL
LIN {X 0,Y 326.168,Z 1179.928,A -85,B 0,C 180,E1 15176.655,E2 15176.655} C_VEL
LIN {X 0,Y 331.061,Z 1164.179,A -85,B 0,C 180,E1 15174.132,E2 15174.132} C_VEL
LIN {X 0,Y 335.645,Z 1148.183,A -85,B 0,C 180,E1 15172.021,E2 15172.021} C_VEL
LIN {X 0,Y 340.114,Z 1130.841,A -85,B 0,C 180,E1 15170.143,E2 15170.143} C_VEL
LIN {X 0,Y 344.232,Z 1112.381,A -85,B 0,C 180,E1 15168.528,E2 15168.528} C_VEL
LIN {X 0,Y 347.649,Z 1094.043,A -85,B 0,C 180,E1 15167.253,E2 15167.253} C_VEL
LIN {X 0,Y 350.583,Z 1074.243,A -85,B 0,C 180,E1 15166.18,E2 15166.18} C_VEL
